# B&R Automation Studio project ABC_Pltzr (part 5)

#### appDraw.typ - Local data types
```iecst
TYPE
	paDrawEnums_typ :
		(
		PADRAW_RECT_MAXIDX := 30
		);
	paCallback_typ : 	STRUCT
		pCallback : REFERENCE TO UDINT;
		callbackValue : UDINT;
		callbackState : UDINT;
		callbackRet : UDINT;
		callbackParams : ARRAY[0..3]OF UDINT;
	END_STRUCT;
	paDrawBoxSize_typ : 	STRUCT
		name : STRING[31];
		length_inch : REAL; (*Width (pixels) of the draw box control*)
		width_inch : REAL; (*Width (pixels) of the draw box control*)
		height_inch : REAL; (*Height (pixels) of the draw box control*)
		length_pixel : UDINT; (*Width (pixels) of the draw box control*)
		width_pixel : UDINT; (*Width (pixels) of the draw box control*)
		height_pixel : UDINT; (*Height (pixels) of the draw box control*)
	END_STRUCT;
	paDrawBoxCtrl_typ : 	STRUCT
		state : UDINT;
		handle : UDINT; (*VISAPI handle returned from VA_Setup()*)
		nameDrawBoxCtrl : STRING[80]; (*DrawBox name for VA_Attach(). It is string with a following format "pageName/LayerName/drawBoxComponentName"*)
		nameVisu : STRING[20]; (*Visualization object name within the project (i.e."Visu", "Panel", "Hmi", etc)*)
		colorIndex : USINT; (*Background color index*)
		width : UDINT; (*Width (pixels) of the draw box control*)
		height : UDINT; (*Height (pixels) of the draw box control*)
	END_STRUCT;
	paDrawTextout_typ : 	STRUCT
		iEnable : USINT; (*Enable text output*)
		iFontIndex : USINT; (*Text font index*)
		iFColorIndex : USINT; (*Text front color index*)
		iBColorIndex : USINT; (*Data line color index*)
		iX : REAL; (*Text x position*)
		iY : REAL; (*Text y poistion*)
		iText : STRING[80]; (*Number of samples in dataset*)
	END_STRUCT;
	paDrawRect_typ : 	STRUCT
		iEnable : USINT; (*Enable text output*)
		iVCHandle : UDINT; (*Text font index*)
		iX : UINT; (*Text x position*)
		iY : UINT; (*Text y poistion*)
		iWidth : UINT; (*Text x position*)
		iHeight : UINT; (*Text y poistion*)
		iFillColorIndex : USINT; (*Text front color index*)
		iBorderColorIndex : USINT; (*Data line color index*)
	END_STRUCT;
	paDrawDataset_typ : 	STRUCT
		iColorIndex : USINT; (*Data line color index*)
		iMinValue : REAL; (*Min value from the data set > will be displayed at 0% on the graph*)
		iMaxValue : REAL; (*Max value from the data set > will be displayed at 100% on the graph*)
		iSizeDataset : UDINT; (*Number of samples in dataset*)
		ipDataset : REFERENCE TO REAL; (*Reference (pointer) to the dataset*)
	END_STRUCT;
	paDrawBoxGrid_typ : 	STRUCT
		ivColorIndex : USINT; (*Grid line color - vertical line*)
		ivLineCount : USINT; (*Number of vertical lines*)
		ivThickRepeat : USINT; (*Place a thicker (i.e. divider) grid line repeat count times - vertical*)
		ihColorIndex : USINT; (*Grid line color - horizontal line*)
		ihLineCount : USINT; (*Number of horizontal lines*)
		ihThickRepeat : USINT; (*Place a thicker (i.e. divider) grid line repeat count times - horizontal*)
	END_STRUCT;
	paDrawXZMotionProfile_typ : 	STRUCT
		ixPhysicalRange : REAL;
		izPhysicalRange : REAL;
		ixPick : REAL;
		izPick : REAL;
		ixDrop : REAL;
		izDrop : REAL;
		iFwdClrIdx : USINT;
		iRevClrIdx : USINT;
		ixCamDataset : paDrawDataset_typ;
		izCamDataset : paDrawDataset_typ;
		idx : UDINT;
		deltaCamMaster : REAL;
		state : UDINT;
	END_STRUCT;
	paDrawBoxDrawing_typ : 	STRUCT
		cb : paCallback_typ;
		ctrl : paDrawBoxCtrl_typ;
		grid : paDrawBoxGrid_typ;
		rect : paDrawRect_typ;
		textout : paDrawTextout_typ;
		data1 : paDrawDataset_typ;
		pRectArray : REFERENCE TO paDrawRect_typ;
		xzProfile : paDrawXZMotionProfile_typ;
	END_STRUCT;
	paCamEditApp_typ : 	STRUCT
		btnPreview : USINT;
		state : UDINT;
		camPointsX : ARRAY[0..3]OF REAL;
		camPointsZ : ARRAY[0..3]OF REAL;
		value : USINT;
	END_STRUCT;
END_TYPE
```

- bgstring.c (reference to Logical/paiComponents/bglib/bgstring.c)

### Program Logical/MachineControl/animation (IEC) - app animation

#### Variables.var
```iecst
VAR
	jj : UDINT := 0;
	ii : UDINT := 0;
END_VAR
```

#### Cyclic.st
```iecst
PROGRAM _CYCLIC
	(* Insert code here *)

	gCtrlAnimation.tmrCase();

	FOR ii :=0 TO 9 BY 1 DO
		IF ii  <  gCtrlAnimation.currentCase THEN
			gCtrlAnimation.visiCase.animationRow[ii] := 0;//visible
		ELSE
			gCtrlAnimation.visiCase.animationRow[ii] := 1;//not visible
		END_IF;

		IF ii  <  gCtrlAnimation.currentRow THEN
			FOR jj := 0 TO 9 BY 1 DO
				IF jj < gConfigApp.options.dryCycleCaseCount THEN
					gCtrlAnimation.visiRow[ii].animationRow[jj] := 0;//visible
				ELSE
					gCtrlAnimation.visiRow[ii].animationRow[jj] := 1;//not visible
				END_IF;
			END_FOR;

		ELSE
			FOR jj := 0 TO 9 BY 1 DO
				gCtrlAnimation.visiRow[ii].animationRow[jj] := 1;//not visible
			END_FOR;
		END_IF;

		IF ii  <  gCtrlAnimation.currentLayer THEN
			FOR jj := 0 TO 9 BY 1 DO
				IF jj < gConfigApp.options.dryCycleRowCount THEN
					gCtrlAnimation.visiLayer[ii].animationRow[jj] := 0;//visible
				ELSE
					gCtrlAnimation.visiLayer[ii].animationRow[jj] := 1;//not visible
				END_IF;
			END_FOR;

		ELSE
			FOR jj := 0 TO 9 BY 1 DO
				gCtrlAnimation.visiLayer[ii].animationRow[jj] := 1;//not visible
			END_FOR;
		END_IF;

	END_FOR;

	IF ((animationState <> 0) AND (NOT gCtrl.main.noFaults)) THEN
		animationState := 50;
	END_IF;

	CASE animationState OF
		0:
			gCtrlAnimation.currentCase := 0;
			gCtrlAnimation.currentRow := 0;
			gCtrlAnimation.currentLayer := 0;
			IF gCtrl.main.modeAuto THEN
				animationState := 10;
				gCtrl.infeedcv.hmiBtnOnOff := 1;
				gCtrl.rowforming.hmiBtnOnOffCV := 1;
			END_IF;
		10:
			gCtrlAnimation.currentCase := gCtrlAnimation.currentCase + 1;
			IF gCtrlAnimation.currentCase >= gConfigApp.options.dryCycleCaseCount THEN
				gCtrl.rowforming.hmiBtnPusherFwd := 1;
				gCtrl.rowforming.hmiBtnPusherRev := 0;
				gCtrl.infeedcv.hmiBtnOnOff := 0;
				gCtrl.rowforming.hmiBtnOnOffCV := 0;
				animationState := 11;
			ELSE
				animationState := 20;
			END_IF;
		11://waiting for row pusher at elev
			IF gCtrl.rowforming.isRowPusherAtElevator THEN
				gCtrlAnimation.currentCase := 0;
				gCtrlAnimation.currentRow := gCtrlAnimation.currentRow + 1;
				gCtrl.rowforming.hmiBtnPusherFwd := 0;
				gCtrl.rowforming.hmiBtnPusherRev := 1;

				IF gCtrlAnimation.currentRow >= gConfigApp.options.dryCycleRowCount THEN
					gCtrl.main.testBit1 := 1;//start elev drycycle
					animationState := 13;
				ELSE
					animationState := 12;
				END_IF;
			END_IF;
		12://waiting for row pusher back home
			IF gCtrl.rowforming.isRowPusherAtHome THEN
				gCtrl.infeedcv.hmiBtnOnOff := 1;
				gCtrl.rowforming.hmiBtnOnOffCV := 1;

				animationState := 20;
			END_IF;
		13:
			IF gCtrl.main.testBit3 THEN//wait for elev dry cycle to complete
				gCtrl.main.testBit3 := 0;
				animationState := 14;
			END_IF;
		14:
			gCtrlAnimation.currentRow := 0;
			gCtrlAnimation.currentLayer := gCtrlAnimation.currentLayer + 1;
			IF gCtrlAnimation.currentLayer >= gConfigApp.options.dryCycleLayerCount THEN
				animationState := 30;
			ELSE
				gCtrl.infeedcv.hmiBtnOnOff := 1;
				gCtrl.rowforming.hmiBtnOnOffCV := 1;

				animationState := 20;
			END_IF;
		20:
			gCtrl.infeedcv.hmiBtnOnOff := 1;
			gCtrl.rowforming.hmiBtnOnOffCV := 1;
			gCtrlAnimation.tmrCase.IN := 0;
			gCtrlAnimation.tmrCase.PT := REAL_TO_UDINT(gConfigApp.options.tmDryCycleCaseTime * 1000);

			IF (gConfigApp.options.dryCycleCaseCount >= 2) AND  (gCtrlAnimation.currentCase = 1) THEN
				gCtrl.caseturner.hmiBtnCaseTurnerUpDown := 1;	//turn on blade1 and case turner
				gCtrl.rowforming.hmiBtnStopBladeUpDown1 := 1;
			ELSE
				gCtrl.caseturner.hmiBtnCaseTurnerUpDown := 0;
				gCtrl.rowforming.hmiBtnStopBladeUpDown1 := 0;
			END_IF;

			animationState := 21;
			IF gCtrl.main.modeManual THEN
				animationState := 50;
			END_IF;

		21:
			gCtrlAnimation.tmrCase.IN := 1;
			IF gCtrlAnimation.tmrCase.Q THEN
				gCtrlAnimation.tmrCase.IN := 0;
				animationState := 10;
			END_IF;

		30:
			//Pallete is Done!
			IF gConfigApp.options.dryCycleLayerDonePause <> 0 THEN
				gPaiHmiRTMenu.iMenuSelectItem[1] := 1;//switch to manual mode
				gCtrlAnimation.tmrCase.IN := 0;
				gCtrlAnimation.tmrCase.PT := T#1s;
				animationState := 31;
			ELSE
				//continue with a new layer
				animationState := 0;//clear all, and start cycle again
			END_IF;
		31:
			gCtrlAnimation.tmrCase.IN := 1;
			IF gCtrlAnimation.tmrCase.Q THEN
				IF gCtrl.main.modeAuto THEN
					animationState := 0;//clear all, and start cycle again
				END_IF;
			END_IF;

		50:
		//wait for resume
			gCtrl.infeedcv.hmiBtnOnOff := 0;
			gCtrl.rowforming.hmiBtnOnOffCV := 0;
			IF gCtrl.main.modeAuto THEN
				gCtrl.infeedcv.hmiBtnOnOff := 1;
				gCtrl.rowforming.hmiBtnOnOffCV := 1;
				animationState := 20;
			END_IF;

	END_CASE;

END_PROGRAM
```

### Program Logical/MachineControl/alarms (IEC) - app alarms

#### Cyclic.ld
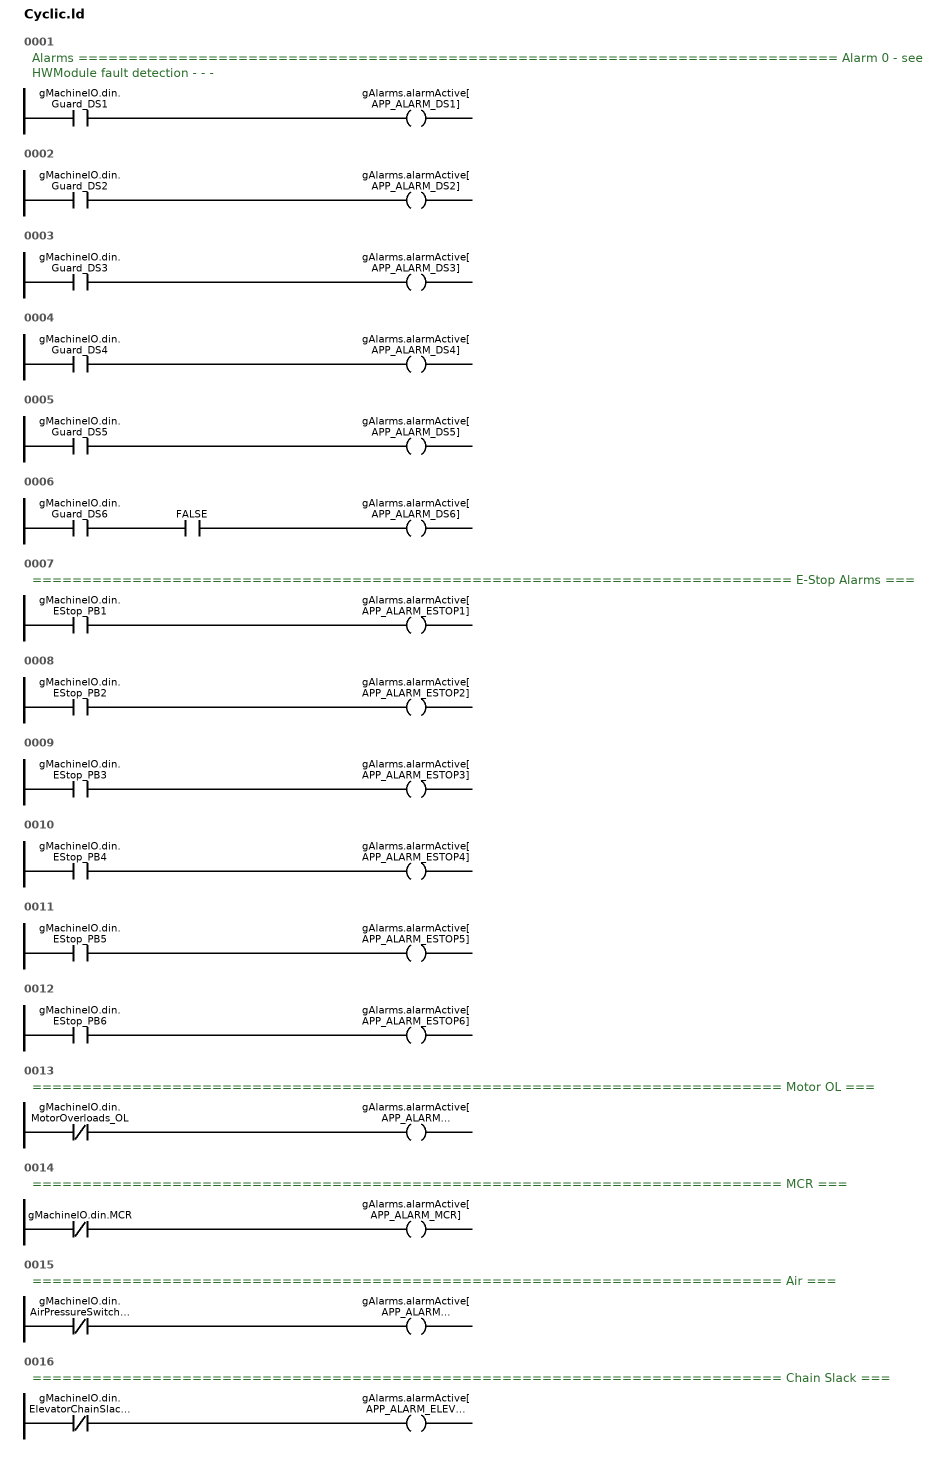
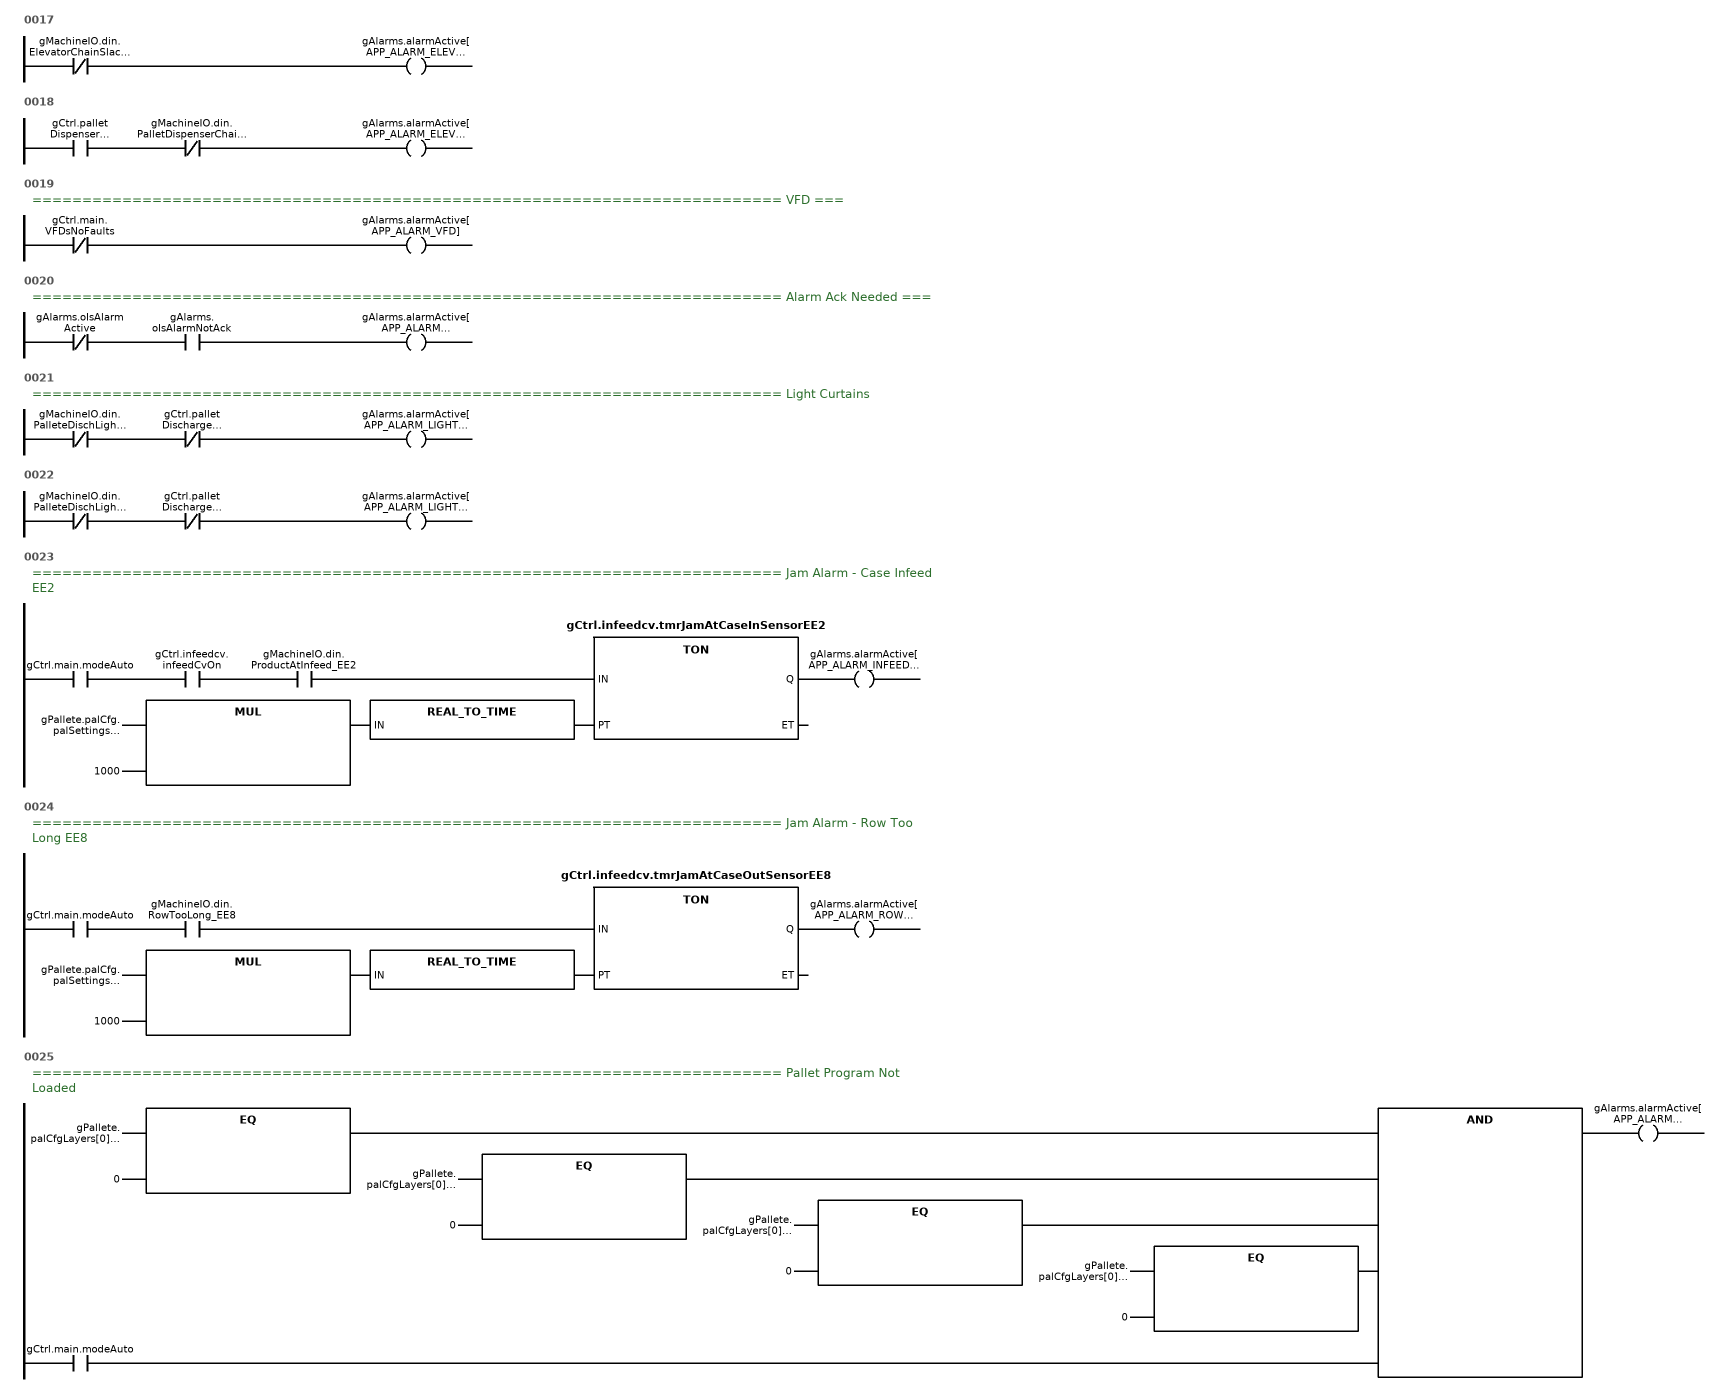
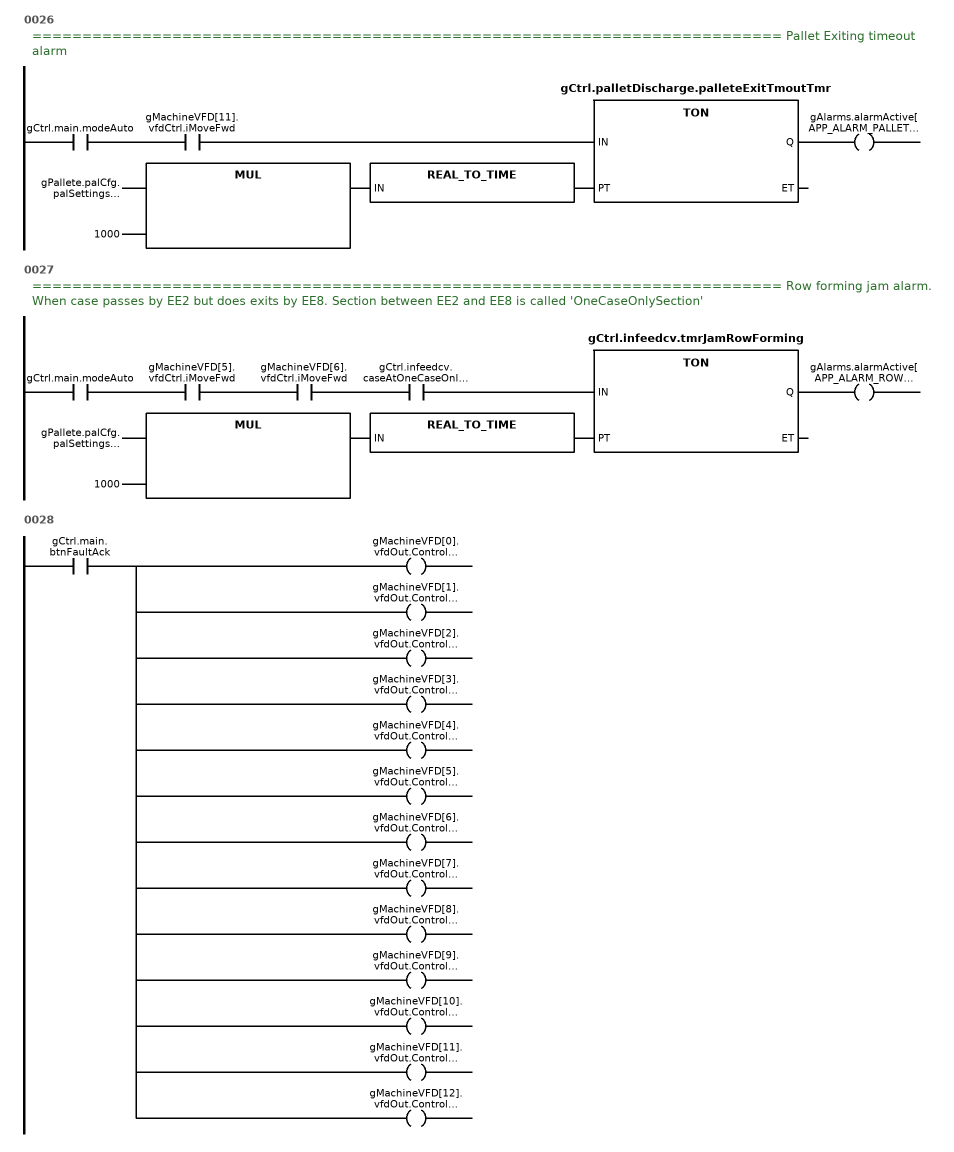
Ladder, written as Structured Text:
```iecst
PROGRAM _CYCLIC
(* Network 1: Alarms ============================================================================ Alarm 0 - see HWModule fault detection - - - *)
gAlarms.alarmActive[APP_ALARM_DS1] := gMachineIO.din.Guard_DS1;

(* Network 2 *)
gAlarms.alarmActive[APP_ALARM_DS2] := gMachineIO.din.Guard_DS2;

(* Network 3 *)
gAlarms.alarmActive[APP_ALARM_DS3] := gMachineIO.din.Guard_DS3;

(* Network 4 *)
gAlarms.alarmActive[APP_ALARM_DS4] := gMachineIO.din.Guard_DS4;

(* Network 5 *)
gAlarms.alarmActive[APP_ALARM_DS5] := gMachineIO.din.Guard_DS5;

(* Network 6 *)
gAlarms.alarmActive[APP_ALARM_DS6] := FALSE;

(* Network 7: ============================================================================ E-Stop Alarms === *)
gAlarms.alarmActive[APP_ALARM_ESTOP1] := gMachineIO.din.EStop_PB1;

(* Network 8 *)
gAlarms.alarmActive[APP_ALARM_ESTOP2] := gMachineIO.din.EStop_PB2;

(* Network 9 *)
gAlarms.alarmActive[APP_ALARM_ESTOP3] := gMachineIO.din.EStop_PB3;

(* Network 10 *)
gAlarms.alarmActive[APP_ALARM_ESTOP4] := gMachineIO.din.EStop_PB4;

(* Network 11 *)
gAlarms.alarmActive[APP_ALARM_ESTOP5] := gMachineIO.din.EStop_PB5;

(* Network 12 *)
gAlarms.alarmActive[APP_ALARM_ESTOP6] := gMachineIO.din.EStop_PB6;

(* Network 13: =========================================================================== Motor OL === *)
gAlarms.alarmActive[APP_ALARM_MOTOROL] := NOT gMachineIO.din.MotorOverloads_OL;

(* Network 14: =========================================================================== MCR === *)
gAlarms.alarmActive[APP_ALARM_MCR] := NOT gMachineIO.din.MCR;

(* Network 15: =========================================================================== Air === *)
gAlarms.alarmActive[APP_ALARM_AIRPRESSURE] := NOT gMachineIO.din.AirPressureSwitch_APS;

(* Network 16: =========================================================================== Chain Slack === *)
gAlarms.alarmActive[APP_ALARM_ELEV_CHAINSLACK_LF] := NOT gMachineIO.din.ElevatorChainSlackLF_LS7;

(* Network 17 *)
gAlarms.alarmActive[APP_ALARM_ELEV_CHAINSLACK_RT] := NOT gMachineIO.din.ElevatorChainSlackRT_LS8;

(* Network 18 *)
gAlarms.alarmActive[APP_ALARM_ELEV_PALLETDISPENS] := gCtrl.palletDispenser.palletDispenserEquipped AND NOT gMachineIO.din.PalletDispenserChainSlack_PR21;

(* Network 19: =========================================================================== VFD === *)
gAlarms.alarmActive[APP_ALARM_VFD] := NOT gCtrl.main.VFDsNoFaults;

(* Network 20: =========================================================================== Alarm Ack Needed === *)
gAlarms.alarmActive[APP_ALARM_ALARMACKNEEDED] := NOT gAlarms.oIsAlarmActive AND gAlarms.oIsAlarmNotAck;

(* Network 21: =========================================================================== Light Curtains *)
gAlarms.alarmActive[APP_ALARM_LIGHT_CURTAIN_OSSD1] := NOT gMachineIO.din.PalleteDischLightCurtain_OSSD1 AND NOT gCtrl.palletDischarge.muteLightCurtainDuringDischarge;

(* Network 22 *)
gAlarms.alarmActive[APP_ALARM_LIGHT_CURTAIN_OSSD2] := NOT gMachineIO.din.PalleteDischLightCurtain_OSSD2 AND NOT gCtrl.palletDischarge.muteLightCurtainDuringDischarge;

(* Network 23: =========================================================================== Jam Alarm - Case Infeed EE2 *)
gCtrl.infeedcv.tmrJamAtCaseInSensorEE2(IN := gCtrl.main.modeAuto AND gCtrl.infeedcv.infeedCvOn AND gMachineIO.din.ProductAtInfeed_EE2, PT := REAL_TO_TIME(gPallete.palCfg.palSettings.timers.JamAlarmTmAtInfeedEE2 * 1000));
gAlarms.alarmActive[APP_ALARM_INFEED_JAM] := gCtrl.infeedcv.tmrJamAtCaseInSensorEE2.Q;

(* Network 24: =========================================================================== Jam Alarm - Row Too Long EE8 *)
gCtrl.infeedcv.tmrJamAtCaseOutSensorEE8(IN := gCtrl.main.modeAuto AND gMachineIO.din.RowTooLong_EE8, PT := REAL_TO_TIME(gPallete.palCfg.palSettings.timers.JamAlarmTmAtRowToLongEE8 * 1000));
gAlarms.alarmActive[APP_ALARM_ROW_TOO_LONG] := gCtrl.infeedcv.tmrJamAtCaseOutSensorEE8.Q;

(* Network 25: =========================================================================== Pallet Program Not Loaded *)
gAlarms.alarmActive[APP_ALARM_INVALID_PROGRAM] := (gPallete.palCfgLayers[0].palCfgRows[0].palCfgCmds[0].cmdCase = 0) AND (gPallete.palCfgLayers[0].palCfgRows[0].palCfgCmds[0].cmdBlade = 0) AND (gPallete.palCfgLayers[0].palCfgRows[0].palCfgCmds[0].cmdFeature = 0) AND (gPallete.palCfgLayers[0].palCfgRows[0].palCfgCmds[0].cmdExtra = 0) AND gCtrl.main.modeAuto;

(* Network 26: =========================================================================== Pallet Exiting timeout alarm *)
gCtrl.palletDischarge.palleteExitTmoutTmr(IN := gCtrl.main.modeAuto AND gMachineVFD[11].vfdCtrl.iMoveFwd, PT := REAL_TO_TIME(gPallete.palCfg.palSettings.timers.palletExitAlarmTm * 1000));
gAlarms.alarmActive[APP_ALARM_PALLET_EXIT_TIMEOUT] := gCtrl.palletDischarge.palleteExitTmoutTmr.Q;

(* Network 27: =========================================================================== Row forming jam alarm. When case passes by EE2 but does exits by EE8. Section between EE2 and EE8 is called 'OneCaseOnlySection' *)
gCtrl.infeedcv.tmrJamRowForming(IN := gCtrl.main.modeAuto AND gMachineVFD[5].vfdCtrl.iMoveFwd AND gMachineVFD[6].vfdCtrl.iMoveFwd AND gCtrl.infeedcv.caseAtOneCaseOnlySection, PT := REAL_TO_TIME(gPallete.palCfg.palSettings.timers.JamAlarmTmRowForming * 1000));
gAlarms.alarmActive[APP_ALARM_ROW_FORMING_JAM] := gCtrl.infeedcv.tmrJamRowForming.Q;

(* Network 28 *)
gMachineVFD[0].vfdOut.Control.FaultReset := gCtrl.main.btnFaultAck;
gMachineVFD[1].vfdOut.Control.FaultReset := gCtrl.main.btnFaultAck;
gMachineVFD[2].vfdOut.Control.FaultReset := gCtrl.main.btnFaultAck;
gMachineVFD[3].vfdOut.Control.FaultReset := gCtrl.main.btnFaultAck;
gMachineVFD[4].vfdOut.Control.FaultReset := gCtrl.main.btnFaultAck;
gMachineVFD[5].vfdOut.Control.FaultReset := gCtrl.main.btnFaultAck;
gMachineVFD[6].vfdOut.Control.FaultReset := gCtrl.main.btnFaultAck;
gMachineVFD[7].vfdOut.Control.FaultReset := gCtrl.main.btnFaultAck;
gMachineVFD[8].vfdOut.Control.FaultReset := gCtrl.main.btnFaultAck;
gMachineVFD[9].vfdOut.Control.FaultReset := gCtrl.main.btnFaultAck;
gMachineVFD[10].vfdOut.Control.FaultReset := gCtrl.main.btnFaultAck;
gMachineVFD[11].vfdOut.Control.FaultReset := gCtrl.main.btnFaultAck;
gMachineVFD[12].vfdOut.Control.FaultReset := gCtrl.main.btnFaultAck;
END_PROGRAM
```

### Program Logical/MachineControl/messages (IEC) - app HMI messages

#### Cyclic.ld
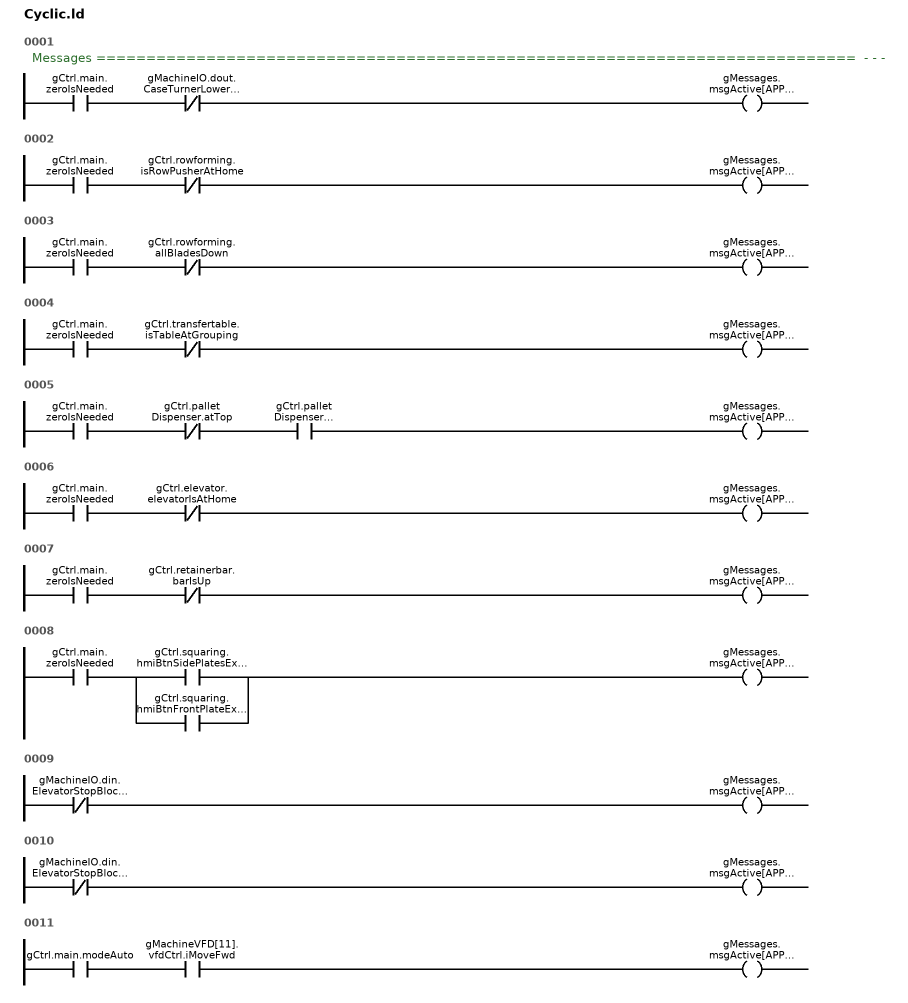
Ladder, written as Structured Text:
```iecst
PROGRAM _CYCLIC
(* Network 1: Messages ============================================================================  - - - *)
gMessages.msgActive[APP_MSG_ZERO_CASETURNER] := gCtrl.main.zeroIsNeeded AND NOT gMachineIO.dout.CaseTurnerLower_SOL2B;

(* Network 2 *)
gMessages.msgActive[APP_MSG_ZERO_ROWPUSHER] := gCtrl.main.zeroIsNeeded AND NOT gCtrl.rowforming.isRowPusherAtHome;

(* Network 3 *)
gMessages.msgActive[APP_MSG_ZERO_BLADESTOP] := gCtrl.main.zeroIsNeeded AND NOT gCtrl.rowforming.allBladesDown;

(* Network 4 *)
gMessages.msgActive[APP_MSG_ZERO_TABLE] := gCtrl.main.zeroIsNeeded AND NOT gCtrl.transfertable.isTableAtGrouping;

(* Network 5 *)
gMessages.msgActive[APP_MSG_ZERO_PALLETELIFT] := gCtrl.main.zeroIsNeeded AND NOT gCtrl.palletDispenser.atTop AND gCtrl.palletDispenser.palletDispenserEquipped;

(* Network 6 *)
gMessages.msgActive[APP_MSG_ZERO_ELEVATOR] := gCtrl.main.zeroIsNeeded AND NOT gCtrl.elevator.elevatorIsAtHome;

(* Network 7 *)
gMessages.msgActive[APP_MSG_ZERO_RETAINERBAR] := gCtrl.main.zeroIsNeeded AND NOT gCtrl.retainerbar.barIsUp;

(* Network 8 *)
gMessages.msgActive[APP_MSG_ZERO_SQUARING] := gCtrl.main.zeroIsNeeded AND (gCtrl.squaring.hmiBtnSidePlatesExtRet OR gCtrl.squaring.hmiBtnFrontPlateExtRet);

(* Network 9 *)
gMessages.msgActive[APP_MSG_STOP_BLOCK_LF] := NOT gMachineIO.din.ElevatorStopBlockLF_PR33;

(* Network 10 *)
gMessages.msgActive[APP_MSG_STOP_BLOCK_RT] := NOT gMachineIO.din.ElevatorStopBlockRT_PR34;

(* Network 11 *)
gMessages.msgActive[APP_MSG_PALLETE_EXITING] := gCtrl.main.modeAuto AND gMachineVFD[11].vfdCtrl.iMoveFwd;
END_PROGRAM
```

### Program Logical/MachineControl/safety (IEC) - app Machine Safety

#### Cyclic.ld
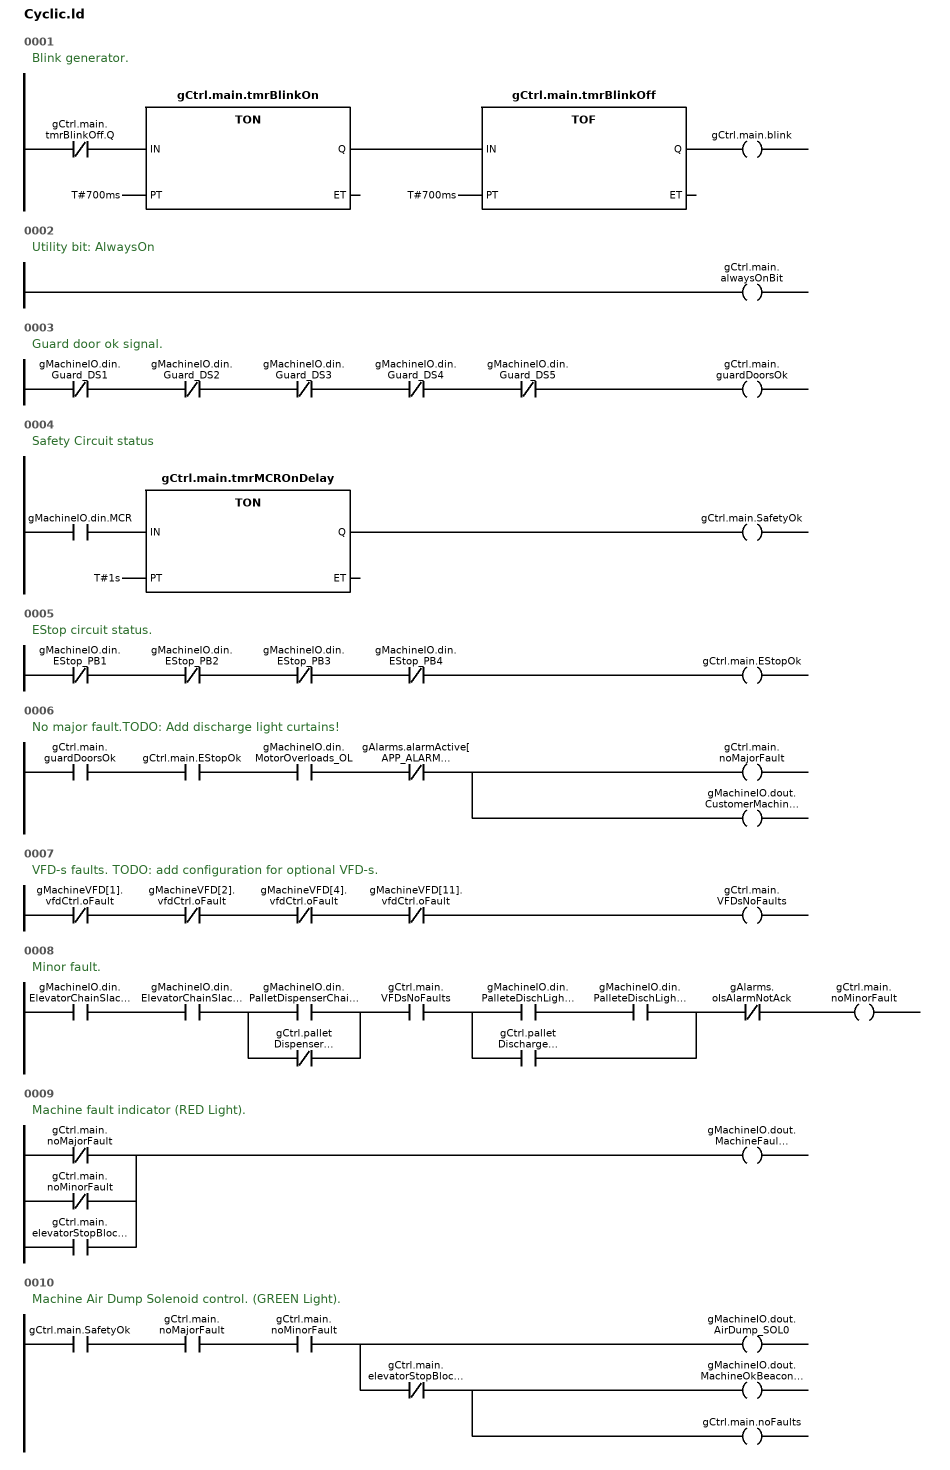
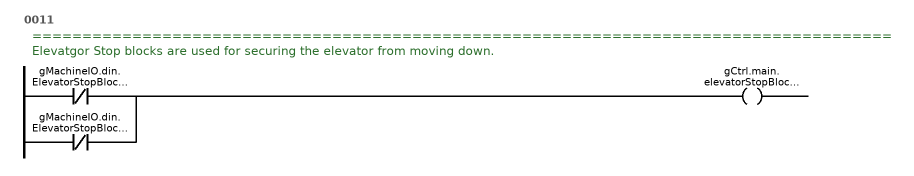
Ladder, written as Structured Text:
```iecst
PROGRAM _CYCLIC
VAR
    _p1 : BOOL;
    _p2 : BOOL;
    _p3 : BOOL;
    _p4 : BOOL;
END_VAR
(* Network 1: Blink generator. *)
gCtrl.main.tmrBlinkOn(IN := NOT gCtrl.main.tmrBlinkOff.Q, PT := T#700ms);
gCtrl.main.tmrBlinkOff(IN := gCtrl.main.tmrBlinkOn.Q, PT := T#700ms);
gCtrl.main.blink := gCtrl.main.tmrBlinkOff.Q;

(* Network 2: Utility bit: AlwaysOn *)
gCtrl.main.alwaysOnBit := TRUE;

(* Network 3: Guard door ok signal. *)
gCtrl.main.guardDoorsOk := NOT gMachineIO.din.Guard_DS1 AND NOT gMachineIO.din.Guard_DS2 AND NOT gMachineIO.din.Guard_DS3 AND NOT gMachineIO.din.Guard_DS4 AND NOT gMachineIO.din.Guard_DS5;

(* Network 4: Safety Circuit status *)
gCtrl.main.tmrMCROnDelay(IN := gMachineIO.din.MCR, PT := T#1s);
gCtrl.main.SafetyOk := gCtrl.main.tmrMCROnDelay.Q;

(* Network 5: EStop circuit status. *)
gCtrl.main.EStopOk := NOT gMachineIO.din.EStop_PB1 AND NOT gMachineIO.din.EStop_PB2 AND NOT gMachineIO.din.EStop_PB3 AND NOT gMachineIO.din.EStop_PB4;

(* Network 6: No major fault.TODO: Add discharge light curtains! *)
_p1 := gCtrl.main.guardDoorsOk AND gCtrl.main.EStopOk AND gMachineIO.din.MotorOverloads_OL AND NOT gAlarms.alarmActive[APP_ALARM_HWMODULE];
gCtrl.main.noMajorFault := _p1;
gMachineIO.dout.CustomerMachineRunning_CR5 := _p1;

(* Network 7: VFD-s faults. TODO: add configuration for optional VFD-s. *)
gCtrl.main.VFDsNoFaults := NOT gMachineVFD[1].vfdCtrl.oFault AND NOT gMachineVFD[2].vfdCtrl.oFault AND NOT gMachineVFD[4].vfdCtrl.oFault AND NOT gMachineVFD[11].vfdCtrl.oFault;

(* Network 8: Minor fault. *)
_p2 := gMachineIO.din.ElevatorChainSlackLF_LS7 AND gMachineIO.din.ElevatorChainSlackRT_LS8;
_p3 := _p2 AND (gMachineIO.din.PalletDispenserChainSlack_PR21 OR NOT gCtrl.palletDispenser.palletDispenserEquipped) AND gCtrl.main.VFDsNoFaults;
gCtrl.main.noMinorFault := _p3 AND ((gMachineIO.din.PalleteDischLightCurtain_OSSD1 AND gMachineIO.din.PalleteDischLightCurtain_OSSD2) OR gCtrl.palletDischarge.muteLightCurtainDuringDischarge) AND NOT gAlarms.oIsAlarmNotAck;

(* Network 9: Machine fault indicator (RED Light). *)
gMachineIO.dout.MachineFaultBeacon_LT1 := NOT gCtrl.main.noMajorFault OR NOT gCtrl.main.noMinorFault OR gCtrl.main.elevatorStopBlockActive;

(* Network 10: Machine Air Dump Solenoid control. (GREEN Light). *)
_p4 := gCtrl.main.SafetyOk AND gCtrl.main.noMajorFault AND gCtrl.main.noMinorFault;
gMachineIO.dout.AirDump_SOL0 := _p4;
gMachineIO.dout.MachineOkBeacon_LT2 := _p4 AND NOT gCtrl.main.elevatorStopBlockActive;
gCtrl.main.noFaults := _p4 AND NOT gCtrl.main.elevatorStopBlockActive;

(* Network 11: ====================================================================================== Elevatgor Stop blocks are used for securing the elevator from moving down. *)
gCtrl.main.elevatorStopBlockActive := NOT gMachineIO.din.ElevatorStopBlockLF_PR33 OR NOT gMachineIO.din.ElevatorStopBlockRT_PR34;
END_PROGRAM
```

### Program Logical/MachineControl/machzero (IEC) - app Machine Zeroing

#### Cyclic.ld
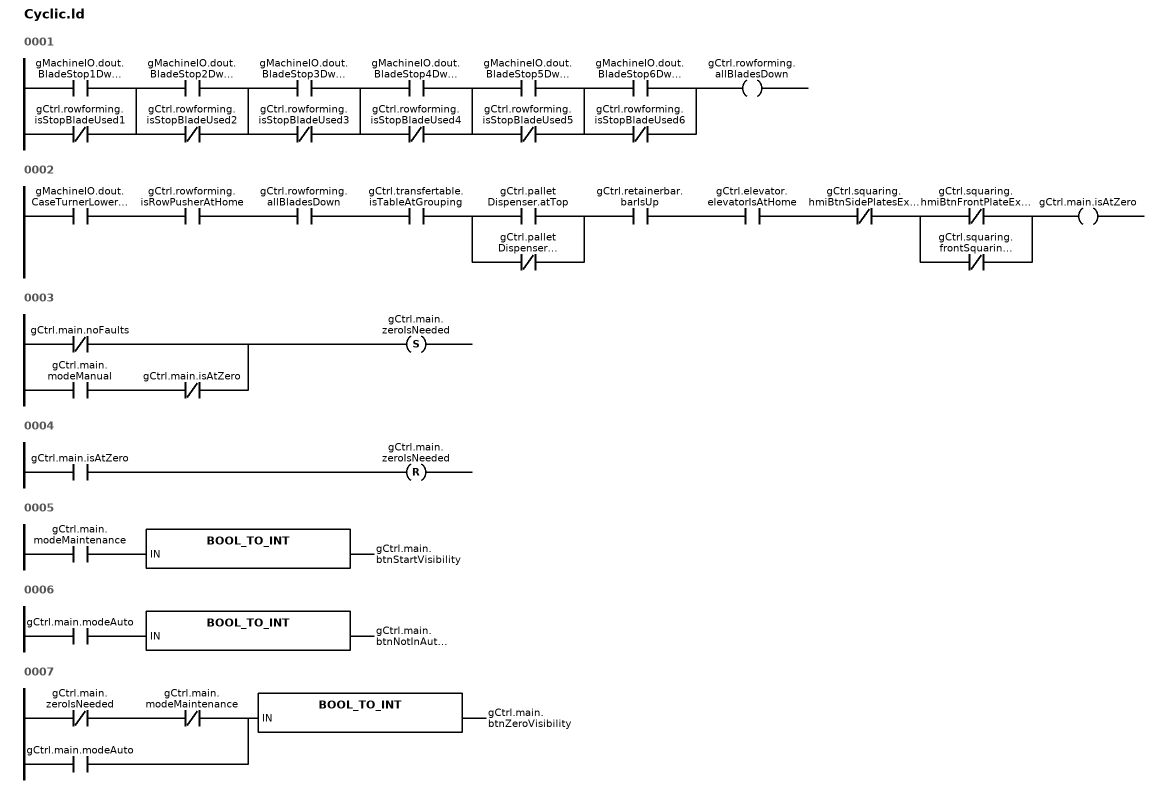
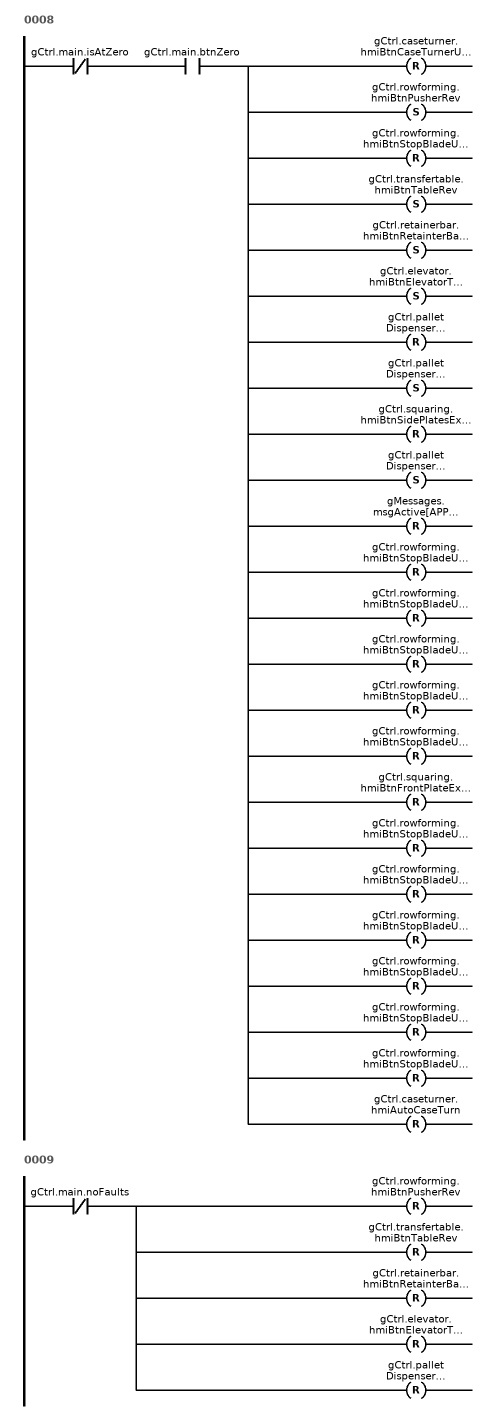
Ladder, written as Structured Text:
```iecst
PROGRAM _CYCLIC
VAR
    _p1 : BOOL;
    _p2 : BOOL;
    _p3 : BOOL;
    _p4 : BOOL;
    _p5 : BOOL;
    _p6 : BOOL;
    _p7 : BOOL;
    _p8 : BOOL;
    _p9 : BOOL;
    _p10 : BOOL;
    _p11 : BOOL;
    _p12 : BOOL;
END_VAR
(* Network 1 *)
_p1 := (gMachineIO.dout.BladeStop1Dw_SOL3B OR NOT gCtrl.rowforming.isStopBladeUsed1) AND gMachineIO.dout.BladeStop2Dw_SOL4B;
_p2 := (gMachineIO.dout.BladeStop1Dw_SOL3B OR NOT gCtrl.rowforming.isStopBladeUsed1) AND NOT gCtrl.rowforming.isStopBladeUsed2;
_p3 := (_p1 OR _p2) AND gMachineIO.dout.BladeStop3Dw_SOL5B;
_p4 := (_p1 OR _p2) AND NOT gCtrl.rowforming.isStopBladeUsed3;
_p5 := (_p3 OR _p4) AND gMachineIO.dout.BladeStop4Dw_SOL6B;
_p6 := (_p3 OR _p4) AND NOT gCtrl.rowforming.isStopBladeUsed4;
_p7 := (_p5 OR _p6) AND gMachineIO.dout.BladeStop5Dw_SOL13B;
_p8 := (_p5 OR _p6) AND NOT gCtrl.rowforming.isStopBladeUsed5;
gCtrl.rowforming.allBladesDown := (_p7 OR _p8) AND (gMachineIO.dout.BladeStop6Dw_SOL14B OR NOT gCtrl.rowforming.isStopBladeUsed6);

(* Network 2 *)
_p9 := gMachineIO.dout.CaseTurnerLower_SOL2B AND gCtrl.rowforming.isRowPusherAtHome AND gCtrl.rowforming.allBladesDown AND gCtrl.transfertable.isTableAtGrouping;
_p10 := _p9 AND (gCtrl.palletDispenser.atTop OR NOT gCtrl.palletDispenser.palletDispenserEquipped) AND gCtrl.retainerbar.barIsUp AND gCtrl.elevator.elevatorIsAtHome AND NOT gCtrl.squaring.hmiBtnSidePlatesExtRet;
gCtrl.main.isAtZero := _p10 AND (NOT gCtrl.squaring.hmiBtnFrontPlateExtRet OR NOT gCtrl.squaring.frontSquaringEquipped);

(* Network 3 *)
IF NOT gCtrl.main.noFaults OR (gCtrl.main.modeManual AND NOT gCtrl.main.isAtZero) THEN
    gCtrl.main.zeroIsNeeded := TRUE;
END_IF;

(* Network 4 *)
IF gCtrl.main.isAtZero THEN gCtrl.main.zeroIsNeeded := FALSE; END_IF;

(* Network 5 *)
gCtrl.main.btnStartVisibility := BOOL_TO_INT(gCtrl.main.modeMaintenance);

(* Network 6 *)
gCtrl.main.btnNotInAutoModeVisibility := BOOL_TO_INT(gCtrl.main.modeAuto);

(* Network 7 *)
gCtrl.main.btnZeroVisibility := BOOL_TO_INT((NOT gCtrl.main.zeroIsNeeded AND NOT gCtrl.main.modeMaintenance) OR gCtrl.main.modeAuto);

(* Network 8 *)
_p11 := NOT gCtrl.main.isAtZero AND gCtrl.main.btnZero;
IF NOT gCtrl.main.isAtZero AND gCtrl.main.btnZero THEN
    gCtrl.caseturner.hmiBtnCaseTurnerUpDown := FALSE;
END_IF;
IF _p11 THEN
    gCtrl.rowforming.hmiBtnPusherRev := TRUE;
    gCtrl.rowforming.hmiBtnStopBladeUpDown1 := FALSE;
    gCtrl.transfertable.hmiBtnTableRev := TRUE;
    gCtrl.retainerbar.hmiBtnRetainterBarRev := TRUE;
    gCtrl.elevator.hmiBtnElevatorToGrouping := TRUE;
    gCtrl.palletDispenser.hmiBtnPalletClawsOpenClose := FALSE;
    gCtrl.palletDispenser.hmiBtnClawsLiftToTop := TRUE;
    gCtrl.squaring.hmiBtnSidePlatesExtRet := FALSE;
    gCtrl.palletDispenser.hmiBtnPalletClawsOpenClose := TRUE;
    gMessages.msgActive[APP_MSG_PALLETE_COMPLETE] := FALSE;
    gCtrl.rowforming.hmiBtnStopBladeUpDown2 := FALSE;
    gCtrl.rowforming.hmiBtnStopBladeUpDown3 := FALSE;
    gCtrl.rowforming.hmiBtnStopBladeUpDown4 := FALSE;
    gCtrl.rowforming.hmiBtnStopBladeUpDown5 := FALSE;
    gCtrl.rowforming.hmiBtnStopBladeUpDown6 := FALSE;
    gCtrl.squaring.hmiBtnFrontPlateExtRet := FALSE;
    gCtrl.rowforming.hmiBtnStopBladeUpDownQuick1 := FALSE;
    gCtrl.rowforming.hmiBtnStopBladeUpDownQuick2 := FALSE;
    gCtrl.rowforming.hmiBtnStopBladeUpDownQuick3 := FALSE;
    gCtrl.rowforming.hmiBtnStopBladeUpDownQuick4 := FALSE;
    gCtrl.rowforming.hmiBtnStopBladeUpDownQuick5 := FALSE;
    gCtrl.rowforming.hmiBtnStopBladeUpDownQuick6 := FALSE;
    gCtrl.caseturner.hmiAutoCaseTurn := FALSE;
END_IF;

(* Network 9 *)
_p12 := NOT gCtrl.main.noFaults;
IF NOT gCtrl.main.noFaults THEN gCtrl.rowforming.hmiBtnPusherRev := FALSE; END_IF;
IF _p12 THEN
    gCtrl.transfertable.hmiBtnTableRev := FALSE;
    gCtrl.retainerbar.hmiBtnRetainterBarRev := FALSE;
    gCtrl.elevator.hmiBtnElevatorToGrouping := FALSE;
    gCtrl.palletDispenser.hmiBtnClawsLiftToTop := FALSE;
END_IF;
END_PROGRAM
```

- Program Logical/MachineControl/infcvidle (IEC) - app infeed CV idle logic (no source held here)

### Program Logical/MachineControl/rowforming (IEC) - app row forming

#### Cyclic.ld - Cyclic code
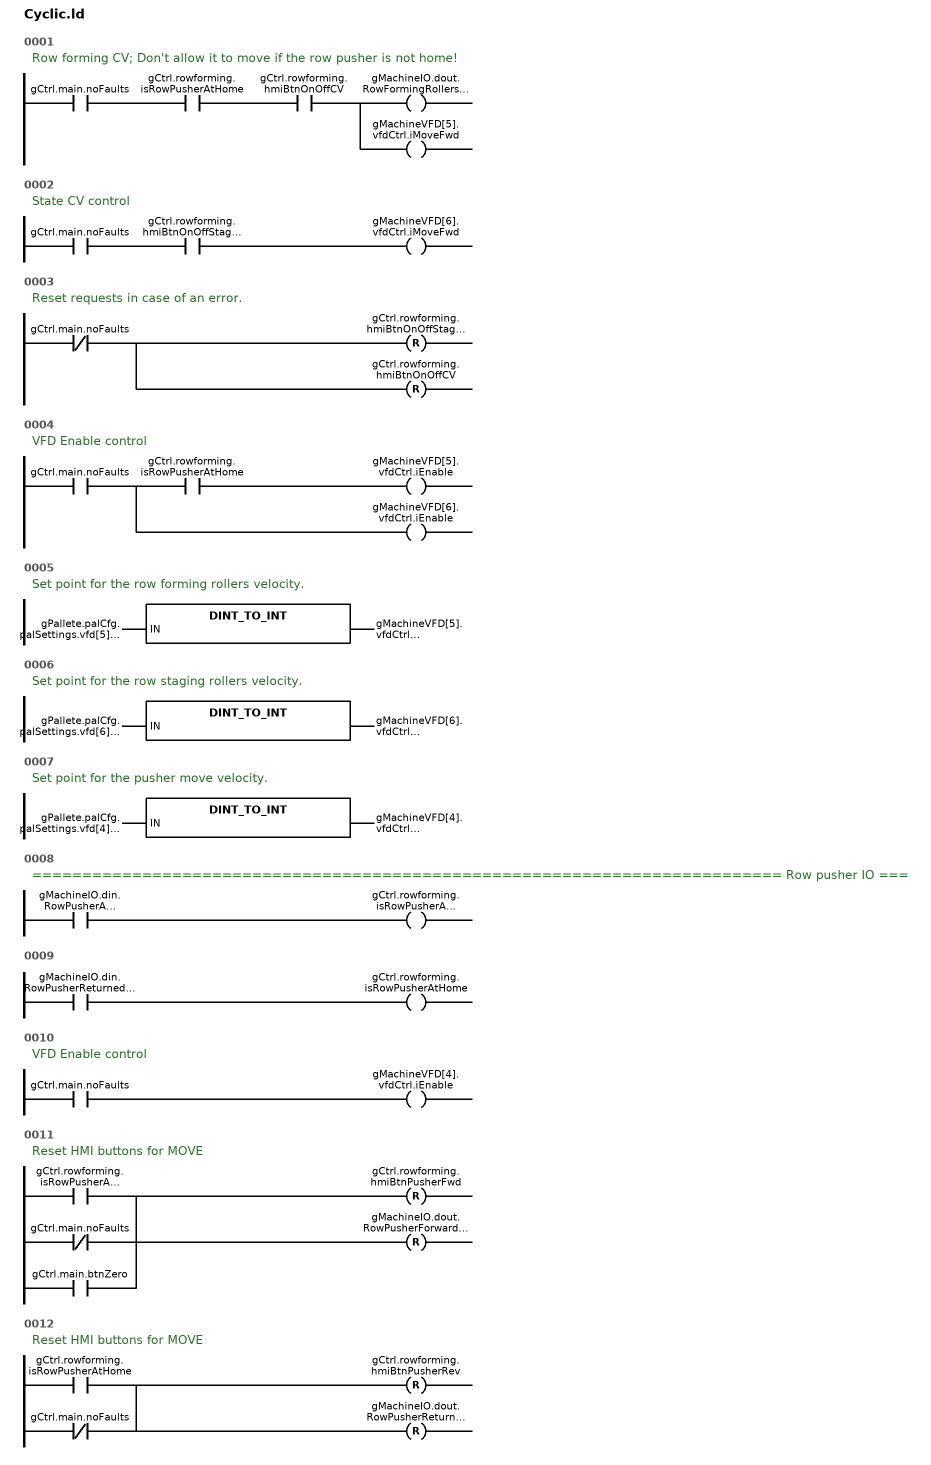
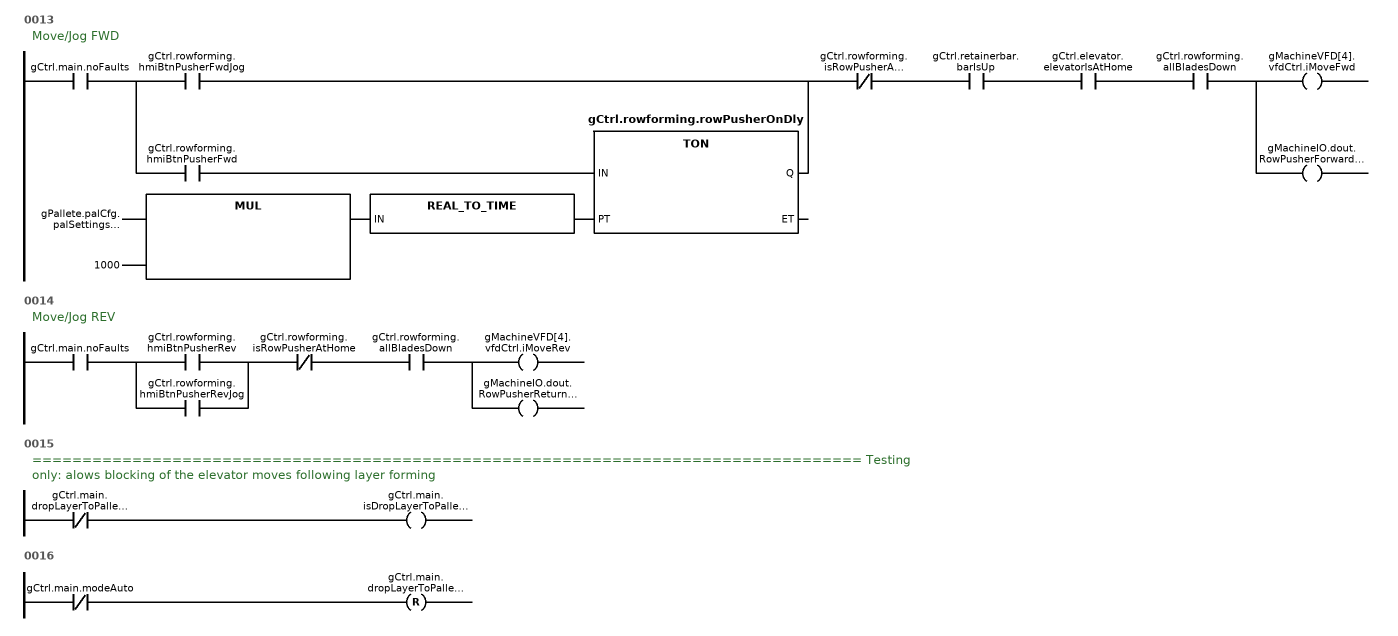
Ladder, written as Structured Text:
```iecst
PROGRAM _CYCLIC
VAR
    _p1 : BOOL;
    _p2 : BOOL;
    _p3 : BOOL;
    _p4 : BOOL;
    _p5 : BOOL;
    _p6 : BOOL;
    _p7 : BOOL;
    _p8 : BOOL;
    _p9 : BOOL;
END_VAR
(* Network 1: Row forming CV; Don't allow it to move if the row pusher is not home! *)
_p1 := gCtrl.main.noFaults AND gCtrl.rowforming.isRowPusherAtHome AND gCtrl.rowforming.hmiBtnOnOffCV;
gMachineIO.dout.RowFormingRollers_M5 := _p1;
gMachineVFD[5].vfdCtrl.iMoveFwd := _p1;

(* Network 2: State CV control *)
gMachineVFD[6].vfdCtrl.iMoveFwd := gCtrl.main.noFaults AND gCtrl.rowforming.hmiBtnOnOffStageCV;

(* Network 3: Reset requests in case of an error. *)
_p2 := NOT gCtrl.main.noFaults;
IF NOT gCtrl.main.noFaults THEN gCtrl.rowforming.hmiBtnOnOffStageCV := FALSE; END_IF;
IF _p2 THEN gCtrl.rowforming.hmiBtnOnOffCV := FALSE; END_IF;

(* Network 4: VFD Enable control *)
gMachineVFD[5].vfdCtrl.iEnable := gCtrl.main.noFaults AND gCtrl.rowforming.isRowPusherAtHome;
gMachineVFD[6].vfdCtrl.iEnable := gCtrl.main.noFaults;

(* Network 5: Set point for the row forming rollers velocity. *)
gMachineVFD[5].vfdCtrl.iVelocitySetPoint := DINT_TO_INT(gPallete.palCfg.palSettings.vfd[5].velocity_rpm);

(* Network 6: Set point for the row staging rollers velocity. *)
gMachineVFD[6].vfdCtrl.iVelocitySetPoint := DINT_TO_INT(gPallete.palCfg.palSettings.vfd[6].velocity_rpm);

(* Network 7: Set point for the pusher move velocity. *)
gMachineVFD[4].vfdCtrl.iVelocitySetPoint := DINT_TO_INT(gPallete.palCfg.palSettings.vfd[4].velocity_rpm);

(* Network 8: =========================================================================== Row pusher IO === *)
gCtrl.rowforming.isRowPusherAtElevator := gMachineIO.din.RowPusherAtElevator_PR13;

(* Network 9 *)
gCtrl.rowforming.isRowPusherAtHome := gMachineIO.din.RowPusherReturned_PR11;

(* Network 10: VFD Enable control *)
gMachineVFD[4].vfdCtrl.iEnable := gCtrl.main.noFaults;

(* Network 11: Reset HMI buttons for MOVE *)
_p3 := gCtrl.rowforming.isRowPusherAtElevator;
_p4 := NOT gCtrl.main.noFaults;
_p5 := gCtrl.main.btnZero;
IF gCtrl.rowforming.isRowPusherAtElevator OR NOT gCtrl.main.noFaults OR gCtrl.main.btnZero THEN
    gCtrl.rowforming.hmiBtnPusherFwd := FALSE;
END_IF;
IF _p3 OR _p4 OR _p5 THEN gMachineIO.dout.RowPusherForward_M4F := FALSE; END_IF;

(* Network 12: Reset HMI buttons for MOVE *)
_p6 := gCtrl.rowforming.isRowPusherAtHome;
_p7 := NOT gCtrl.main.noFaults;
IF gCtrl.rowforming.isRowPusherAtHome OR NOT gCtrl.main.noFaults THEN
    gCtrl.rowforming.hmiBtnPusherRev := FALSE;
END_IF;
IF _p6 OR _p7 THEN gMachineIO.dout.RowPusherReturn_M4R := FALSE; END_IF;

(* Network 13: Move/Jog FWD *)
_p8 := ((gCtrl.main.noFaults AND gCtrl.rowforming.hmiBtnPusherFwdJog) OR gCtrl.rowforming.rowPusherOnDly.Q) AND NOT gCtrl.rowforming.isRowPusherAtElevator AND gCtrl.retainerbar.barIsUp AND gCtrl.elevator.elevatorIsAtHome AND gCtrl.rowforming.allBladesDown;
gMachineVFD[4].vfdCtrl.iMoveFwd := _p8;
gCtrl.rowforming.rowPusherOnDly(IN := gCtrl.main.noFaults AND gCtrl.rowforming.hmiBtnPusherFwd, PT := REAL_TO_TIME(gPallete.palCfg.palSettings.timers.dlyRowDoneToRowPush * 1000));
gMachineIO.dout.RowPusherForward_M4F := _p8;

(* Network 14: Move/Jog REV *)
_p9 := gCtrl.main.noFaults AND (gCtrl.rowforming.hmiBtnPusherRev OR gCtrl.rowforming.hmiBtnPusherRevJog) AND NOT gCtrl.rowforming.isRowPusherAtHome AND gCtrl.rowforming.allBladesDown;
gMachineVFD[4].vfdCtrl.iMoveRev := _p9;
gMachineIO.dout.RowPusherReturn_M4R := _p9;

(* Network 15: =================================================================================== Testing only: alows blocking of the elevator moves following layer forming *)
gCtrl.main.isDropLayerToPalletAllowed := NOT gCtrl.main.dropLayerToPalletBlock;

(* Network 16 *)
IF NOT gCtrl.main.modeAuto THEN gCtrl.main.dropLayerToPalletBlock := FALSE; END_IF;
END_PROGRAM
```

### Program Logical/MachineControl/transtable (IEC) - app transfer table

#### Cyclic.ld
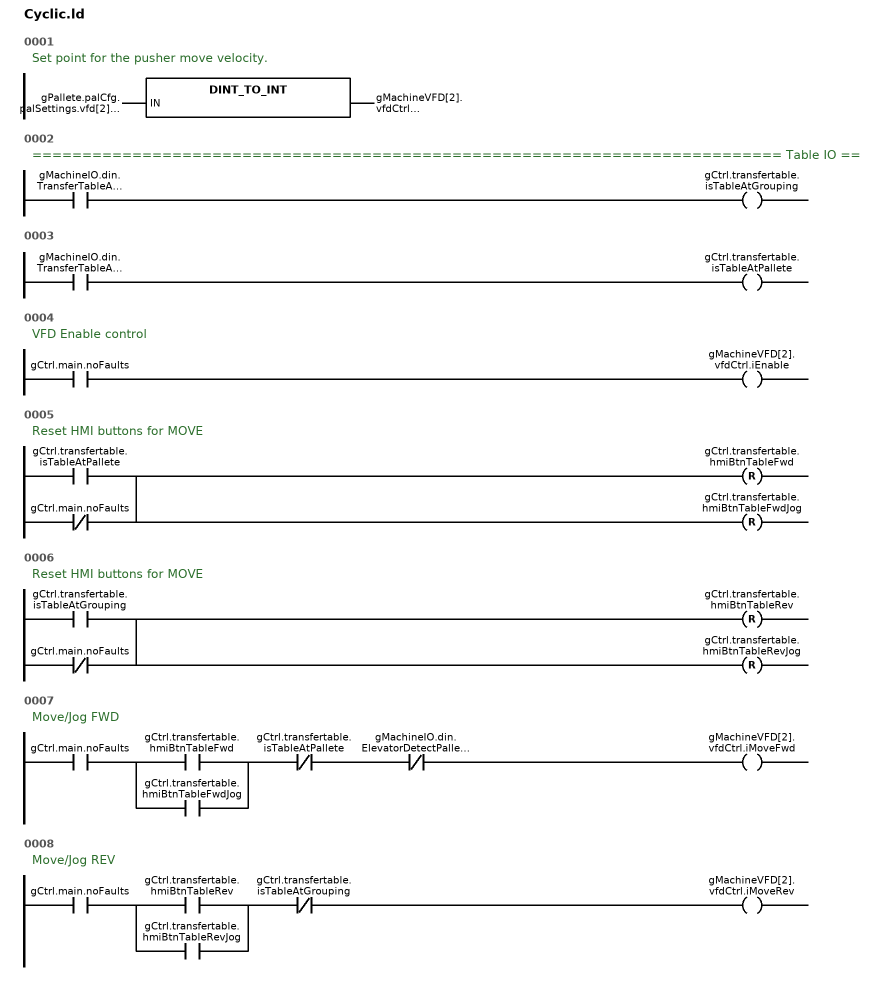
Ladder, written as Structured Text:
```iecst
PROGRAM _CYCLIC
VAR
    _p1 : BOOL;
    _p2 : BOOL;
    _p3 : BOOL;
    _p4 : BOOL;
END_VAR
(* Network 1: Set point for the pusher move velocity. *)
gMachineVFD[2].vfdCtrl.iVelocitySetPoint := DINT_TO_INT(gPallete.palCfg.palSettings.vfd[2].velocity_rpm);

(* Network 2: =========================================================================== Table IO == *)
gCtrl.transfertable.isTableAtGrouping := gMachineIO.din.TransferTableAtGrouping_PR6;

(* Network 3 *)
gCtrl.transfertable.isTableAtPallete := gMachineIO.din.TransferTableAtPallete_PR5;

(* Network 4: VFD Enable control *)
gMachineVFD[2].vfdCtrl.iEnable := gCtrl.main.noFaults;

(* Network 5: Reset HMI buttons for MOVE *)
_p1 := gCtrl.transfertable.isTableAtPallete;
_p2 := NOT gCtrl.main.noFaults;
IF gCtrl.transfertable.isTableAtPallete OR NOT gCtrl.main.noFaults THEN
    gCtrl.transfertable.hmiBtnTableFwd := FALSE;
END_IF;
IF _p1 OR _p2 THEN gCtrl.transfertable.hmiBtnTableFwdJog := FALSE; END_IF;

(* Network 6: Reset HMI buttons for MOVE *)
_p3 := gCtrl.transfertable.isTableAtGrouping;
_p4 := NOT gCtrl.main.noFaults;
IF gCtrl.transfertable.isTableAtGrouping OR NOT gCtrl.main.noFaults THEN
    gCtrl.transfertable.hmiBtnTableRev := FALSE;
END_IF;
IF _p3 OR _p4 THEN gCtrl.transfertable.hmiBtnTableRevJog := FALSE; END_IF;

(* Network 7: Move/Jog FWD *)
gMachineVFD[2].vfdCtrl.iMoveFwd := gCtrl.main.noFaults AND (gCtrl.transfertable.hmiBtnTableFwd OR gCtrl.transfertable.hmiBtnTableFwdJog) AND NOT gCtrl.transfertable.isTableAtPallete AND NOT gMachineIO.din.ElevatorDetectPalletLayerLF_EE1;

(* Network 8: Move/Jog REV *)
gMachineVFD[2].vfdCtrl.iMoveRev := gCtrl.main.noFaults AND (gCtrl.transfertable.hmiBtnTableRev OR gCtrl.transfertable.hmiBtnTableRevJog) AND NOT gCtrl.transfertable.isTableAtGrouping;
END_PROGRAM
```

### Program Logical/MachineControl/palletinfcv (IEC) - app pallet infeed conveyer

#### Cyclic.ld
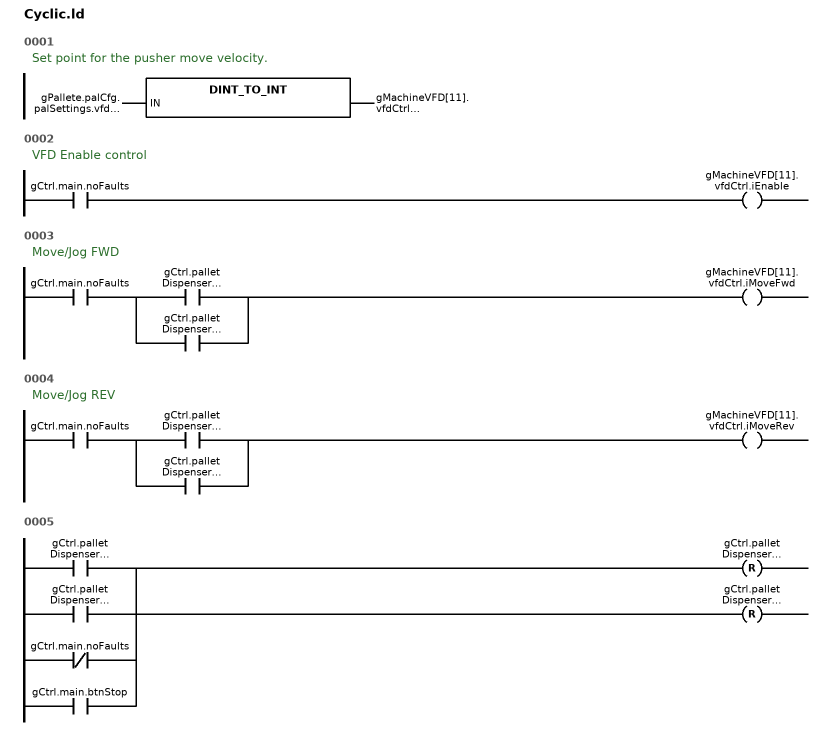
Ladder, written as Structured Text:
```iecst
PROGRAM _CYCLIC
VAR
    _p1 : BOOL;
    _p2 : BOOL;
    _p3 : BOOL;
    _p4 : BOOL;
END_VAR
(* Network 1: Set point for the pusher move velocity. *)
gMachineVFD[11].vfdCtrl.iVelocitySetPoint := DINT_TO_INT(gPallete.palCfg.palSettings.vfd[11].velocity_rpm);

(* Network 2: VFD Enable control *)
gMachineVFD[11].vfdCtrl.iEnable := gCtrl.main.noFaults;

(* Network 3: Move/Jog FWD *)
gMachineVFD[11].vfdCtrl.iMoveFwd := gCtrl.main.noFaults AND (gCtrl.palletDispenser.hmiBtnPalletInCVFwd OR gCtrl.palletDispenser.hmiBtnPalletInCVFwdJog);

(* Network 4: Move/Jog REV *)
gMachineVFD[11].vfdCtrl.iMoveRev := gCtrl.main.noFaults AND (gCtrl.palletDispenser.hmiBtnPalletInCVRev OR gCtrl.palletDispenser.hmiBtnPalletInCVRevJog);

(* Network 5 *)
_p1 := gCtrl.palletDispenser.hmiBtnPalletInCVRevJog;
_p2 := gCtrl.palletDispenser.hmiBtnPalletInCVFwdJog;
_p3 := NOT gCtrl.main.noFaults;
_p4 := gCtrl.main.btnStop;
IF gCtrl.palletDispenser.hmiBtnPalletInCVRevJog OR gCtrl.palletDispenser.hmiBtnPalletInCVFwdJog OR NOT gCtrl.main.noFaults OR gCtrl.main.btnStop THEN
    gCtrl.palletDispenser.hmiBtnPalletInCVFwd := FALSE;
END_IF;
IF _p1 OR _p2 OR _p3 OR _p4 THEN gCtrl.palletDispenser.hmiBtnPalletInCVRev := FALSE; END_IF;
END_PROGRAM
```

### Program Logical/MachineControl/palletinfauto (IEC) - app pallete infeed dispenser auto logic

#### Cyclic.st
```iecst
PROGRAM _CYCLIC
	(* Insert code here *)
	gCtrl.palletDispenser.clawsOpenTmr();

	IF ((gCtrl.palletDispenser.dispenseState <> 0) AND (NOT gCtrl.main.noFaults)) THEN
		gCtrl.palletDispenser.dispenseState := 0;
	END_IF;

	CASE gCtrl.palletDispenser.dispenseState OF

		PLT_DISPENSE_ZERO :
			IF gCtrl.main.modeAuto THEN//wait here for auto mode
				gCtrl.palletDispenser.dispenseState := PLT_DISPENSE_INIT;
				gCtrl.palletDispenser.hmiBtnClawsLiftToTop := 1;
			END_IF;

		PLT_DISPENSE_INIT: //make sure to start at top
			IF gCtrl.palletDispenser.atTop THEN
				gCtrl.palletDispenser.hmiBtnPalletClawsOpenClose := 1;//CLOSE CLAWS
				gCtrl.palletDispenser.dispenseState := PLT_DISPENSE_IDLE;
				gCtrl.palletDispenser.dispenseDN := FALSE;
				gCtrl.palletDispenser.dispenseIP := FALSE;
				gCtrl.palletDispenser.dispenseReq := FALSE;
			END_IF;

		PLT_DISPENSE_IDLE:

			gCtrl.palletDispenser.dispenseDN := FALSE;
			gCtrl.palletDispenser.dispenseIP := FALSE;

			IF gCtrl.palletDispenser.dispenseReq THEN
				gCtrl.palletDispenser.dispenseIP := TRUE;
				gCtrl.palletDispenser.hmiBtnClawsLiftToBottom := 1;//GO TO BOTTOM
				gCtrl.palletDispenser.dispenseState := PLT_DISPENSE_TOBOTTOM;
			END_IF;

		PLT_DISPENSE_TOBOTTOM://wait to bottom
			IF gCtrl.palletDispenser.atBottom THEN//WAIT TO GET TO BOTTOM
				gCtrl.palletDispenser.hmiBtnPalletClawsOpenClose := 0;//OPEN CLAWS
				gCtrl.palletDispenser.clawsOpenTmr.IN := 0;
				gCtrl.palletDispenser.clawsOpenTmr.PT := T#3s;
				gCtrl.palletDispenser.dispenseState := PLT_DISPENSE_WTCLAWSOPN;
			END_IF;

		PLT_DISPENSE_WTCLAWSOPN://WAIT FOR CLAWS TO OPEN
			gCtrl.palletDispenser.clawsOpenTmr.IN := 1;
			IF gCtrl.palletDispenser.clawsOpenTmr.Q THEN
				gCtrl.palletDispenser.hmiBtnClawsLiftToMidLo := 1;//move to MID low
				gCtrl.palletDispenser.dispenseState := PLT_DISPENSE_TOMID;
			END_IF;

		PLT_DISPENSE_TOMID://WAIT FOR MID POSITION
			IF gCtrl.palletDispenser.atMidLo THEN//Wait for At mit Low
				gCtrl.palletDispenser.hmiBtnPalletClawsOpenClose := 1;//CLOSE CLAWS

				gCtrl.palletDispenser.clawsOpenTmr.IN := 0;
				gCtrl.palletDispenser.clawsOpenTmr.PT := T#3s;
				gCtrl.palletDispenser.dispenseState := PLT_DISPENSE_WTCLAWSCLS;
			END_IF;

		PLT_DISPENSE_WTCLAWSCLS://WAIT FOR CLAWS TO CLOSE
			gCtrl.palletDispenser.clawsOpenTmr.IN := 1;
			IF gCtrl.palletDispenser.clawsOpenTmr.Q THEN
				gCtrl.palletDispenser.hmiBtnClawsLiftToTop := 1;
				gCtrl.palletDispenser.dispenseState := PLT_DISPENSE_DN;
			END_IF;

		PLT_DISPENSE_DN://END OF DISPENSE CYCLE
			IF gCtrl.palletDispenser.atTop THEN
				gCtrl.palletDispenser.dispenseDN := TRUE;
				gCtrl.palletDispenser.dispenseReq := FALSE;
				gCtrl.palletDispenser.dispenseState := PLT_DISPENSE_IDLE;
			END_IF;

		ELSE

	END_CASE;

END_PROGRAM
```

### Program Logical/MachineControl/palletdischarge (IEC) - app pallet discharge conveyer

#### Cyclic.ld
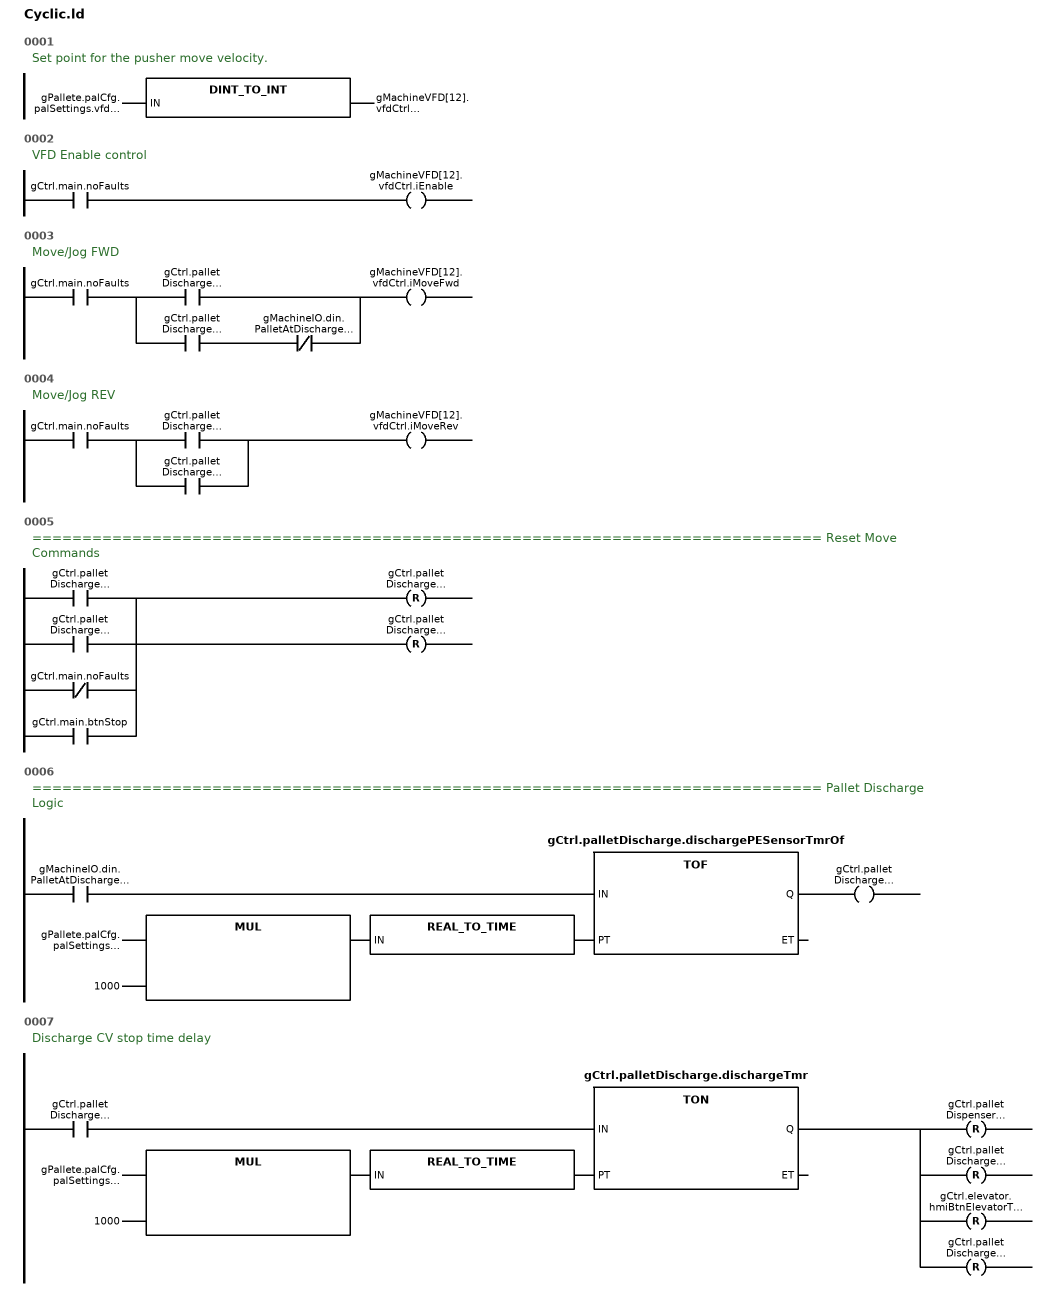
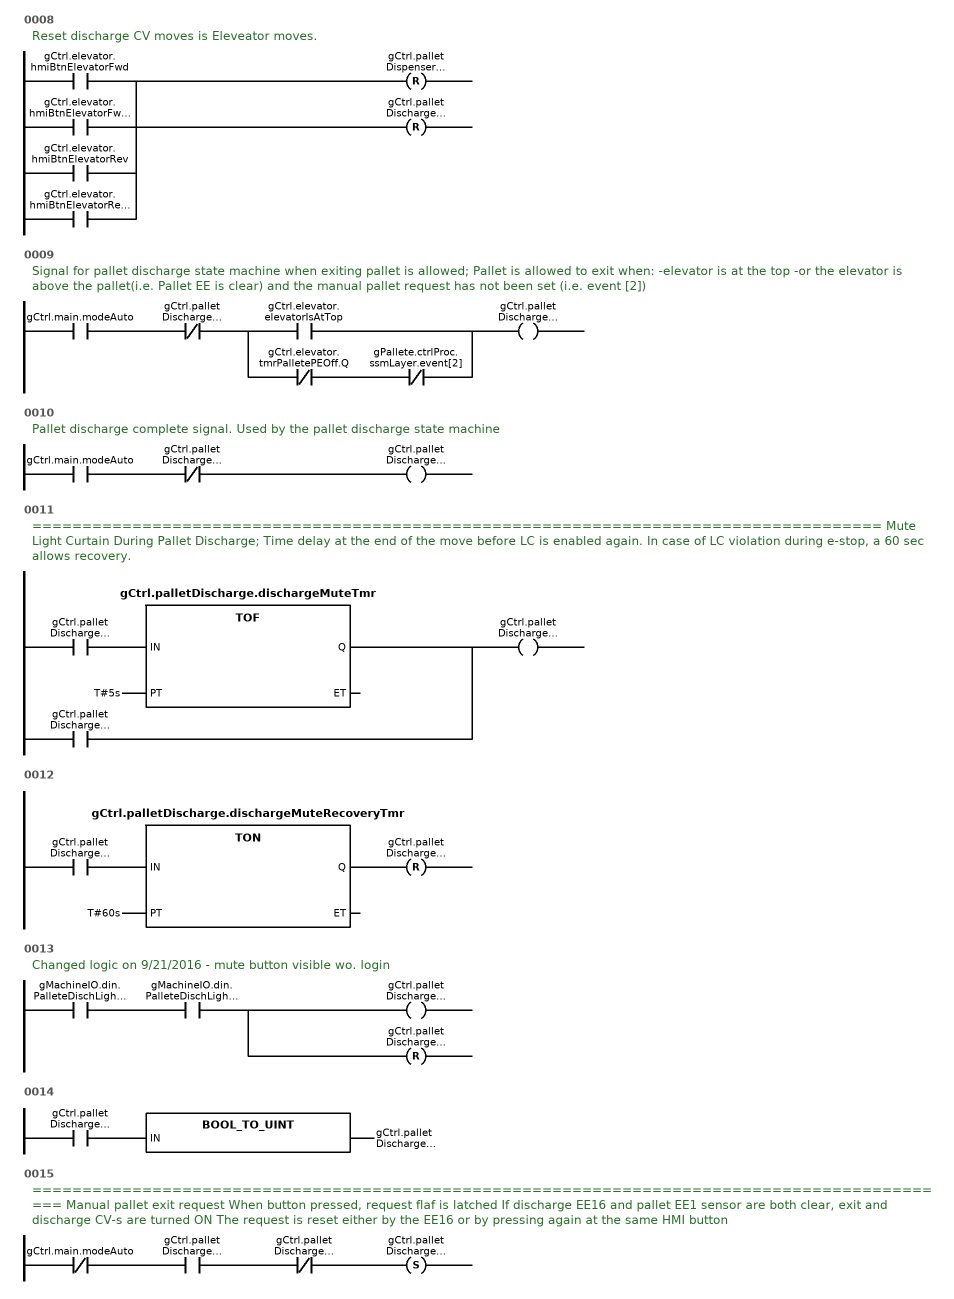
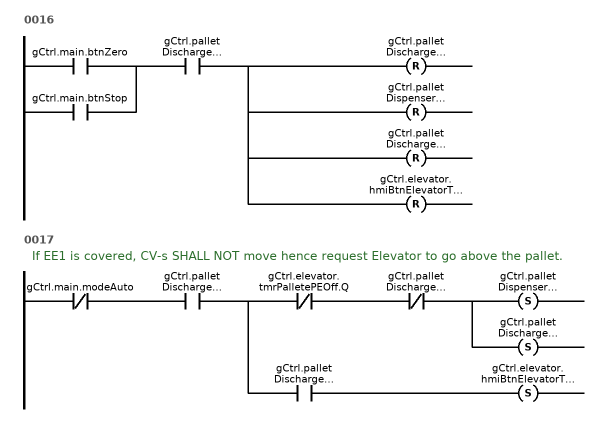
Ladder, written as Structured Text:
```iecst
PROGRAM _CYCLIC
VAR
    _p1 : BOOL;
    _p2 : BOOL;
    _p3 : BOOL;
    _p4 : BOOL;
    _p5 : BOOL;
    _p6 : BOOL;
    _p7 : BOOL;
    _p8 : BOOL;
    _p9 : BOOL;
    _p10 : BOOL;
    _p11 : BOOL;
    _p12 : BOOL;
    _p13 : BOOL;
    _p14 : BOOL;
END_VAR
(* Network 1: Set point for the pusher move velocity. *)
gMachineVFD[12].vfdCtrl.iVelocitySetPoint := DINT_TO_INT(gPallete.palCfg.palSettings.vfd[12].velocity_rpm);

(* Network 2: VFD Enable control *)
gMachineVFD[12].vfdCtrl.iEnable := gCtrl.main.noFaults;

(* Network 3: Move/Jog FWD *)
gMachineVFD[12].vfdCtrl.iMoveFwd := gCtrl.main.noFaults AND (gCtrl.palletDischarge.hmiBtnPalletDischargeCVFwd OR (gCtrl.palletDischarge.hmiBtnPalletDischargeCVFwdJog AND NOT gMachineIO.din.PalletAtDischarge_EE16));

(* Network 4: Move/Jog REV *)
gMachineVFD[12].vfdCtrl.iMoveRev := gCtrl.main.noFaults AND (gCtrl.palletDischarge.hmiBtnPalletDischargeCVRev OR gCtrl.palletDischarge.hmiBtnPalletDischargeCVRevJog);

(* Network 5: =============================================================================== Reset Move Commands *)
_p1 := gCtrl.palletDischarge.hmiBtnPalletDischargeCVRevJog;
_p2 := gCtrl.palletDischarge.hmiBtnPalletDischargeCVFwdJog;
_p3 := NOT gCtrl.main.noFaults;
_p4 := gCtrl.main.btnStop;
IF _p1 OR _p2 OR NOT gCtrl.main.noFaults OR gCtrl.main.btnStop THEN
    gCtrl.palletDischarge.hmiBtnPalletDischargeCVFwd := FALSE;
END_IF;
IF _p1 OR _p2 OR _p3 OR _p4 THEN gCtrl.palletDischarge.hmiBtnPalletDischargeCVRev := FALSE; END_IF;

(* Network 6: =============================================================================== Pallet Discharge Logic *)
gCtrl.palletDischarge.dischargePESensorTmrOf(IN := gMachineIO.din.PalletAtDischarge_EE16, PT := REAL_TO_TIME(gPallete.palCfg.palSettings.timers.EE16OfDebounce * 1000));
gCtrl.palletDischarge.dischargePESensor := gCtrl.palletDischarge.dischargePESensorTmrOf.Q;

(* Network 7: Discharge CV stop time delay *)
gCtrl.palletDischarge.dischargeTmr(IN := gCtrl.palletDischarge.dischargePESensor, PT := REAL_TO_TIME(gPallete.palCfg.palSettings.timers.onDlyPalleteDischargeEE16 * 1000));
_p5 := gCtrl.palletDischarge.dischargeTmr.Q;
IF gCtrl.palletDischarge.dischargeTmr.Q THEN gCtrl.palletDispenser.hmiBtnPalletInCVFwd := FALSE; END_IF;
IF _p5 THEN
    gCtrl.palletDischarge.hmiBtnPalletDischargeCVFwd := FALSE;
    gCtrl.elevator.hmiBtnElevatorToAbovePallete := FALSE;
    gCtrl.palletDischarge.palletManualExitRequest := FALSE;
END_IF;

(* Network 8: Reset discharge CV moves is Eleveator moves. *)
_p6 := gCtrl.elevator.hmiBtnElevatorFwd;
_p7 := gCtrl.elevator.hmiBtnElevatorFwdJog;
_p8 := gCtrl.elevator.hmiBtnElevatorRev;
_p9 := gCtrl.elevator.hmiBtnElevatorRevJog;
IF gCtrl.elevator.hmiBtnElevatorFwd OR gCtrl.elevator.hmiBtnElevatorFwdJog OR gCtrl.elevator.hmiBtnElevatorRev OR gCtrl.elevator.hmiBtnElevatorRevJog THEN
    gCtrl.palletDispenser.hmiBtnPalletInCVFwd := FALSE;
END_IF;
IF _p6 OR _p7 OR _p8 OR _p9 THEN gCtrl.palletDischarge.hmiBtnPalletDischargeCVFwd := FALSE; END_IF;

(* Network 9: Signal for pallet discharge state machine when exiting pallet is allowed; Pallet is allowed to exit when: -elevator is at the top -or the elevator is above the pallet(i.e. Pallet EE is clear) and the manual pallet request has not been set (i.e. event [2]) *)
_p10 := gCtrl.main.modeAuto AND NOT gCtrl.palletDischarge.dischargePESensor;
gCtrl.palletDischarge.isDischargeAllowed := _p10 AND (gCtrl.elevator.elevatorIsAtTop OR (NOT gCtrl.elevator.tmrPalletePEOff.Q AND NOT gPallete.ctrlProc.ssmLayer.event[2]));

(* Network 10: Pallet discharge complete signal. Used by the pallet discharge state machine *)
gCtrl.palletDischarge.dischargeDN := gCtrl.main.modeAuto AND NOT gCtrl.palletDischarge.hmiBtnPalletDischargeCVFwd;

(* Network 11: ===================================================================================== Mute Light Curtain During Pallet Discharge; Time delay at the end of the move before LC is enabled again. In case of LC violation during e-stop, a 60 sec allows recovery. *)
gCtrl.palletDischarge.dischargeMuteTmr(IN := gCtrl.palletDischarge.hmiBtnPalletDischargeCVFwd, PT := T#5s);
gCtrl.palletDischarge.muteLightCurtainDuringDischarge := gCtrl.palletDischarge.dischargeRecoveryIP OR gCtrl.palletDischarge.dischargeMuteTmr.Q;

(* Network 12 *)
gCtrl.palletDischarge.dischargeMuteRecoveryTmr(IN := gCtrl.palletDischarge.dischargeRecoveryIP, PT := T#60s);
IF gCtrl.palletDischarge.dischargeMuteRecoveryTmr.Q THEN
    gCtrl.palletDischarge.dischargeRecoveryIP := FALSE;
END_IF;

(* Network 13: Changed logic on 9/21/2016 - mute button visible wo. login  *)
_p11 := gMachineIO.din.PalleteDischLightCurtain_OSSD1 AND gMachineIO.din.PalleteDischLightCurtain_OSSD2;
gCtrl.palletDischarge.dischargeRecoveryVisible2 := _p11;
IF _p11 THEN gCtrl.palletDischarge.dischargeRecoveryIP := FALSE; END_IF;

(* Network 14 *)
gCtrl.palletDischarge.dischargeRecoveryVisible := BOOL_TO_UINT(gCtrl.palletDischarge.dischargeRecoveryVisible2);

(* Network 15: ============================================================================================= Manual pallet exit request When button pressed, request flaf is latched If discharge EE16 and pallet EE1 sensor are both clear, exit and discharge CV-s are turned ON The request is reset either by the EE16 or by pressing again at the same HMI button *)
IF NOT gCtrl.main.modeAuto AND gCtrl.palletDischarge.hmiBtnPalletManualExit AND NOT gCtrl.palletDischarge.palletManualExitRequest THEN
    gCtrl.palletDischarge.palletManualExitRequest := TRUE;
END_IF;

(* Network 16 *)
_p12 := (gCtrl.main.btnZero OR gCtrl.main.btnStop) AND gCtrl.palletDischarge.palletManualExitRequest;
IF _p12 THEN
    gCtrl.palletDischarge.palletManualExitRequest := FALSE;
    gCtrl.palletDispenser.hmiBtnPalletInCVFwd := FALSE;
    gCtrl.palletDischarge.hmiBtnPalletDischargeCVFwd := FALSE;
    gCtrl.elevator.hmiBtnElevatorToAbovePallete := FALSE;
END_IF;

(* Network 17: If EE1 is covered, CV-s SHALL NOT move hence request Elevator to go above the pallet. *)
_p13 := NOT gCtrl.main.modeAuto AND gCtrl.palletDischarge.palletManualExitRequest;
_p14 := _p13 AND NOT gCtrl.elevator.tmrPalletePEOff.Q AND NOT gCtrl.palletDischarge.dischargePESensor;
IF _p14 THEN
    gCtrl.palletDispenser.hmiBtnPalletInCVFwd := TRUE;
    gCtrl.palletDischarge.hmiBtnPalletDischargeCVFwd := TRUE;
END_IF;
IF _p13 AND gCtrl.palletDischarge.dischargePESensor THEN
    gCtrl.elevator.hmiBtnElevatorToAbovePallete := TRUE;
END_IF;
END_PROGRAM
```

### Program Logical/MachineControl/drycycle (IEC) - app dry cycle machine

#### Variables.var
```iecst
VAR
	elevatorTimer : TON := (0);
END_VAR
```

#### Cyclic.st
```iecst
PROGRAM _CYCLIC
	(* Insert code here *)
	elevatorTimer();

	IF ((dryCycleState <> 0) AND (NOT gCtrl.main.noFaults)) THEN
		dryCycleState := 0;
	END_IF;

	CASE dryCycleState OF
		0 : IF gCtrl.main.testBit1 THEN//wait here
				gCtrl.main.testBit1 := 0;
				dryCycleState := 1;
				elevatorTimer.IN := 0;
				elevatorTimer.PT := REAL_TO_UDINT(gPallete.palCfg.palSettings.timers.dlyTableLayerRdyToElevMove * 1000);
			END_IF;
		1: //wait a delay before start moving elevator
			elevatorTimer.IN := 1;
			IF elevatorTimer.Q THEN
				dryCycleState := 20;
				gCtrl.elevator.hmiBtnElevatorFwd := 1;//move elevator
				elevatorTimer.IN := 0;
				elevatorTimer.PT := REAL_TO_UDINT(gConfigApp.options.tmDryCycleElevatorUp * 1000) * gCtrlAnimation.currentLayer + REAL_TO_UDINT(gConfigApp.options.tmDryCycleLayerZeroOffset * 1000);
			END_IF;

		20://box pusher is done
			elevatorTimer.IN := 1;
			IF elevatorTimer.Q THEN
				elevatorTimer.IN := 0;
				gCtrl.elevator.hmiBtnElevatorFwd := 0;
				gCtrl.transfertable.hmiBtnTableFwd := 1;
				dryCycleState := 30;
			END_IF;
		30:
			IF gCtrl.transfertable.isTableAtPallete THEN
				gCtrl.squaring.hmiBtnSidePlatesExtRet := 1;
				gCtrl.retainerbar.hmiBtnRetainterBarFwd := 1;

				elevatorTimer.IN := 1;
				elevatorTimer.PT := T#3s;

				dryCycleState := 35;
			END_IF;
		35:
			IF elevatorTimer.Q THEN
				gCtrl.transfertable.hmiBtnTableRev := 1;
				dryCycleState := 40;
			END_IF;

		40://
			IF gCtrl.transfertable.isTableAtGrouping THEN
				gCtrl.squaring.hmiBtnSidePlatesExtRet := 0;
				gCtrl.retainerbar.hmiBtnRetainterBarRev := 1;
				gCtrl.elevator.hmiBtnElevatorToGrouping := 1;
				dryCycleState := 50;
			END_IF;
		50://wait for elevator to come back home
			IF gCtrl.elevator.elevatorIsAtHome THEN
				dryCycleState := 0;
				gCtrl.main.testBit3 := 1;
			END_IF;
		60://dry cycle is done

		ELSE

	END_CASE;

END_PROGRAM
```

### Program Logical/MachineControl/drycypal (IEC) - app dry pallete

#### Variables.var
```iecst
VAR
	palleteTimer : TON := (0);
END_VAR
```

### Package Logical/Simulation - application simulation and testing tasks and logic

### Program Logical/Simulation/counter

#### counter.c
```c
/********************************************************************
 * COPYRIGHT -- HP
 ********************************************************************
 * Program: counter
 * File: counter.c
 * Author: goran
 * Created: March 07, 2013
 ********************************************************************
 * Implementation of program counter
 ********************************************************************/

#include <bur/plctypes.h>

#ifdef _DEFAULT_INCLUDES
	#include <AsDefault.h>
#endif

_LOCAL int counter;

void _INIT counterINIT(void)
{
	/* TODO: Add code here */
}

void _CYCLIC counterCYCLIC(void)
{
	/* TODO: Add code here */
	counter++;
	counter++;

}
```

### Program Logical/Simulation/IOsim (ANSIC)

#### IOsim.c - Cyclic code
```c
/********************************************************************
 * COPYRIGHT -- Gainco
 ********************************************************************
 * Program: IO
 * File: IO.c
 * Author: DavidT
 * Created: July 13, 2010
 ********************************************************************
 * Implementation of program IO
 ********************************************************************/

#include <bur/plctypes.h>

#ifdef _DEFAULT_INCLUDES
#include <AsDefault.h>
#endif

#include <..\globalvar.h>
#include <..\..\GlobalDef.h>
#include <..\..\GlobalDecl.h>
//#include "..\\..\\RecFIFO\\fifotest\\fifoif.h"
#include "..\\..\\bglib\\bgsprintf.h"
#include "..\\..\\bglib\\bgsprintf.c"

_LOCAL  BOOL   _inZeroSensor; //n-1 value
_LOCAL  BOOL   _inBeltFlite;  //n-1 value

/*
###############################################################################
Utilities
###############################################################################
*/

/**
 Simple logging
 Log goes to an array of PV strings > see _LOCAL STRING log[][] variable below
 Log output is visible via Automation Studio watch window
 Example of a log statement used within the code is:
 DBG(lgr, "This is log example. %d ", value1);
 To complety disable logging from this source file, change next line to: #if 0
IMPORTANT:
==========
DBGINIT() statement MUST BE PLACED as a first statement within the task _INIT function!
Example:
void _INIT myTaskINIT(void)
{
	//TODO: Add code here
	//init logger object
	DBGINIT(lgr, log, LOG_ENTRY_COUNT, LOG_ENTRY_LENGTH);
}
*/
#if 1
#include <../../bglib/bgPVLogger.c>
#define LOG_ENTRY_COUNT 20	//max number of log entries
#define LOG_ENTRY_LENGTH  32 //max length of individual log message. Longer msg are truncated
_LOCAL STRING log[LOG_ENTRY_COUNT][LOG_ENTRY_LENGTH]; //log output visible from Automation Studio!
static bgPVLogger_typ lgr;	//PV logger object
#else
#define DBG(loggerInstance, format, args...) ;
#define DBGINIT(loggerInstance, logoutput, logEntryCount, logEntrySize)  ;
#endif

#define TK_CYCLE_TIME_Xms 0.01
#define TK_CYCLE_TIME_counts 10
//stage hopper gate control functions for all hoppers
static void stageHoppersGatesClose()
{
	int i;
	for (i=0; i<Config.Cfg_NumTakeoffs; i++)
	{
		Stage[i] = 1;//1 (energized) keeps the gates closed
	}
}

static void stageHoppersGatesOpen()
{
	int i;
	for (i=0; i<Config.Cfg_NumTakeoffs; i++)
	{
		Stage[i] = 0; //0 (not energized) keeps the gates open
	}
}

static BOOL isQCRequiredCurrentStation()
{
	if (QCbypass[OutfeedStation-1] || ((qc[0].QCLoginedIn == 0) && (qc[1].QCLoginedIn == 0)) )
		return 0;//not required when: not request by the HMI and both QC station are not logged in

	return 1;
}

//Find if QC required for the pocket that's going to be dropped next into the outfeed hopper
//OutfeedStation contains number (i.e. 1..16) of the outfeed station that's currently beeing
//dumped into the outfeed hopper (note that it starts with 1 not with 0!)
//
static BOOL isQCRequiredNextStation()
{
int outfeedStationIndexCurrent;
int outfeedStationIndexNext;

	//if OutfeedStation == 0 > no dumping into the outfeed, we are in the search for
	//zero tab > nothing to do
	if(!OutfeedStation)
		return 0;

	//find index (0 based) of the station beeing dumped into the outfeed hopper
	outfeedStationIndexCurrent = OutfeedStation - 1;

	//check if station that's comming next shall be QC-ed
	if(outfeedStationIndexCurrent){
		outfeedStationIndexNext = outfeedStationIndexCurrent - 1;
		if (QCbypass[outfeedStationIndexNext] || (qc[0].QCLoginedIn == 0) )
			return 0;
	}

	//note that for the last station (i.e. OutfeedStation==1), the next station # is Config.Cfg_NumTakeoffs
	if(!outfeedStationIndexCurrent){
		outfeedStationIndexNext = Config.Cfg_NumTakeoffs - 1;
		if (QCbypass[outfeedStationIndexNext] || (qc[0].QCLoginedIn == 0) )
			return 0;
	}

	return 1;
}

//q - qc station index (0 or 1)
static BOOL isQCInspectionActive(int q)
{
	//check if QC inspection is active
	if (qc[q].QCStarted && qc[q].QCLoginedIn)
		return 1;

	return 0;
}

static BOOL isQCLogged_NotStarted(int q)
{
	//check if QC inspection is active
	if (!qc[q].QCStarted && qc[q].QCLoginedIn)
		return 1;

	return 0;
}

//Advance outfeed to the next station
static void outfeedAdvance()
{
	QCselect[0] = 0;
	QCselect[1] = 0;
	if (OutfeedStation == 1)
	{
		ZeroFlag = 0;
		OutfeedStation = 0;
		outstate = 12;
	}
	else
	{
		BeltClutch = 1;
		OutfeedStation--;
		outstate++;
	}

}

//Detect if stopping/pausing outfeed is allowed
static BOOL isOutfeedPauseBlocked()
{
	//Don't allow stop (pause) outfeed SM while belt clutch is on during product indexing
	//That way, we'll avoid a problem with partial dumping of the bin/station content (i.e. if
	//indexing stopped when some product dropped and some product remains in the pocket)
	if( (outstate >= 9) && (outstate <= 11) && BeltClutch )
		return 1; //if above states are active and the belt clutch is on > that's indexing. Don't allow STOP to take place

	//Don't allow stop/pause when the first pocket to be dropped is about to reach the desitnation
	//state 8 is active afer product is dropped onto the belt, until the lead pocket gets dropped into the outfeed hopper
	if( (outstate == 8) && (ZtoDump >= FlightCounter))
		return 1;

	return 0;
}

//Process MasterMode signal and control outfeed state machine
//based upon MasterMode changes
static BOOL outfeedMasterModeLogic()
{
static BOOL _BeltClutch;
static DINT _pauseOperation;
int   i,j;

	//process MasterMode changes
	if (MasterMode != _MasterMode)
	{
		//Previos mode
		switch (_MasterMode)
		{
			case RUN_MODE:
				_BeltClutch = BeltClutch;//preserve belt clutch state when leaving RUN mode
			break;
		}

		//New mode
		switch (MasterMode)
		{
			case STOP_MODE:
				//check if stop/pause is allowed
				if( isOutfeedPauseBlocked() ){
					//pause is blocked, can't switch to stopped mode! wait here until it gets unblocked (i.e. belt turns off)
					//when exiting here, _MasterMode does not get updated. As a result, we'll keep
					//comming back to this point until pause gets unblocked
					return 0;//make sure outfeed SM continues execution!!!
				}

				//entering STOP mode from any other state
				//_BeltClutch = BeltClutch;//preserve belt clutch state
				BeltClutch  = 0;//stop belt
				//NOTE: SM stops executing in this mode, see below
			break;

			case RUN_MODE:
				BeltClutch = _BeltClutch;//restore belt clutch state (preserved when exited RUN state)
				ZeroFlag = 0;//make sure to clear this flag before restoring RUN state

				//when starting RUN from states:
				//0-stopped
				//1-filling
				//3- washdown
				//force the outstate to start at first step in the RUN state (2)
				if(outstate <= 3){
					outstate = 2;
				}else{
					//BAND AID TO MAKE SURE OUTFEED BELT MOVES WHEN SWITCHING TO RUN STATE
					switch(outstate){
						case 5:
						case 6:
						case 8:
						case 9:
						case 11:
							if(!BeltClutch){
								DBG(lgr, "beltOFF,ONreq! otst=%d", outstate);
								BeltClutch = 1;
							}
						break;
					}
				}

				//VERY DIFFICULT PROBLEM DISCOVERED AT MILFORD
				if(outstate == 10){
					OutfeedDumped = 1;//restart handshake to a point that the hopper can pick it up without locking up
				}

				//otherwise, don't touch outstate > it will continue execution from the point where it stopped (outstate > 3)
			break;

			case FILL_MODE:
//				outstate = 1; //start fill
				//check if stop/pause is allowed
				if( isOutfeedPauseBlocked() ){
					//pause is blocked, can't switch to stopped mode! wait here until it gets unblocked (i.e. belt turns off)
					//when exiting here, _MasterMode does not get updated. As a result, we'll keep
					//comming back to this point until pause gets unblocked
					return 0;//make sure outfeed SM continues execution!!!
				}

				//entering STOP mode from any other state
				//_BeltClutch = BeltClutch;//preserve belt clutch state
				BeltClutch  = 0;//stop belt
				//NOTE: SM stops executing in this mode, see below

				//case 1: // fill
					BeltClutch  = 0;
					QCselect[0] = 0;
					QCselect[1] = 0;
					stageHoppersGatesClose();
				//break;

			break;

			case WASHDOWN_MODE:
				outstate = 3; // goto washdown
			break;
		}

		DBG(lgr, "outfeed MasterMode=%d", MasterMode);
		_MasterMode = MasterMode;
	}

	//pause request set
	if(gUdpCmdMsg.outfeed.pauseOperation && !_pauseOperation){
		//same as stop mode
		if(MasterMode == RUN_MODE){

			//check if stop/pause is allowed
			if( isOutfeedPauseBlocked() ){
				//pause is blocked! wait here until it gets unblocked (i.e. belt turns off)
				//when exiting here, _pauseOperation does not get updated. As a result, we'll keep
				//comming back to this point until pause gets unblocked
				return 0;//make sure outfeed SM continues execution!!!
			}

			//pause feature is supported only in RUN mode
			_BeltClutch = BeltClutch;//preserve belt clutch state
			BeltClutch  = 0;//stop belt
		}
		_pauseOperation = gUdpCmdMsg.outfeed.pauseOperation;
	}

	//pause request reset
	if(!gUdpCmdMsg.outfeed.pauseOperation && _pauseOperation){
		if(MasterMode == RUN_MODE){
			//pause feature is supported only in RUN mode
			BeltClutch = _BeltClutch;//restore belt clutch state
			_pauseOperation = gUdpCmdMsg.outfeed.pauseOperation;
		}
	}

	//if STOP mode active > exit here (i.e. don't execute SM)
	if((MasterMode == STOP_MODE) || (MasterMode == FILL_MODE) || (  (MasterMode == RUN_MODE) && _pauseOperation) ){
		return 1;//returning 1 means that outfeed SM will not be executed!!!
	}

	return 0;
}

_LOCAL BOOL lastSelectedQC;

//outfeed state machine
void outfeed(void)
{
int   i,j;
static DINT _OutfeedDumped;

	//process MasterMode and control outfeed SM (outstate)
	//if outfeed SM should be stopped (i.e. not executed, the function returns 1)
	if(outfeedMasterModeLogic()){
		return;
	}

	//log outstate change
	if(outstate != _outstate)
	{
		_outstate = outstate;
		DBG(lgr, "outfeed sm: %d", outstate);
	}

	//log OutfeedDumped change
	if(OutfeedDumped != _OutfeedDumped)
	{
		_OutfeedDumped = OutfeedDumped;
		DBG(lgr, "OfD=%d, Qsl=%d, Qst=%d OfHD=%d", OutfeedDumped, QCselect[0], qc[0].QCStarted, Weigh[1]);

		bgsprintf(gDiagEventRecToFIFO.eventText, "OfD=%d, Qsl=%d, Qst=%d OfHD=%d", OutfeedDumped, QCselect[0], qc[0].QCStarted, Weigh[1]);
		gDiagEventRecToFIFO.eventId = 103;
		captureDiagEvent(gDiagEventRecToFIFO.eventId, gDiagEventRecToFIFO.eventText);
	}

	//outfeed state machine (SM)
	switch (outstate)
	{
	case 0: //stop
		BeltClutch  = 0;
		QCselect[0] = 0;
		QCselect[1] = 0;
		stageHoppersGatesClose();
	break;

	case 1: // fill
		BeltClutch  = 0;
		QCselect[0] = 0;
		QCselect[1] = 0;
		stageHoppersGatesClose();
	break;

	case 2: // run
		//set hw for run
		BeltClutch  = 0;
		QCselect[0] = 0;
		QCselect[1] = 0;
		stageHoppersGatesClose();
		outstate = 4;
	break;

	case 3: // washdown
		// set i/o for washdown
		BeltClutch  = 1;
		QCselect[0] = 0;
		QCselect[1] = 0;
		stageHoppersGatesOpen();
	break;

	case 4: // start outfeed
		BeltClutch = 1;
		outstate++;
	break;

	case 5:  // look for zero tab
		if (ZeroFlag)
		{
			ZeroFlag = 0;
			stop1dly = 0.0;
			outstate++;
		}
	break;

	case 6:  // stop 1 delay after zero tab detected
		stop1dly += .001;
		if (stop1dly > Config.Cfg_Stop1dly)
		{
			BeltClutch = 0;
			ZtoDump = 0;
			Stagedly1 = 0.0;
			Stagedly2 = 0.0;
			stageHoppersGatesOpen();//as soon as the belt stops, dump product onto the outfeed belt
			outstate++;
		}
	break;

	case 7:  // Delay for Dumping Staging Hoppers & dump to outfeed belt

		Stagedly1 += TK_CYCLE_TIME_Xms;
		if (Stagedly1 >= gUdpCmdMsg.outfeed.stagingHopperOpenDuration)
		{
			stageHoppersGatesClose();
//			stageHoppersGatesOpen();

			Stagedly2 += TK_CYCLE_TIME_Xms;
			if (Stagedly2 >= gUdpCmdMsg.outfeed.outfeedBeltCycleStartDelay)
			{
				FltCntFlg  = 0;//reset flight counter
				//stageHoppersGatesClose();
				BeltClutch = 1; // Start Moving belt
				outstate++;
			}
		}
	break;

	case 8:  // Zero to first Dump
		if (FltCntFlg)
		{
			FltCntFlg = 0;
			ZtoDump++;
			if (ZtoDump > FlightCounter)
			{
				stop2dly = 0.0;
				OutfeedStation = Config.Cfg_NumTakeoffs;//set the station that will be processed first at the outfeed hopper
				outstate++;
			}
		}
	break;

	case 9:  // Stop 2 DLY, delay after a flight that contains product that shall be dropped first is detected
		stop2dly += TK_CYCLE_TIME_Xms;
		if (stop2dly > Config.Cfg_Stop2dly)
		{
			BeltClutch = 0;//stop the outfeed belt
			OutfeedDumped = 1;//request to outfeed hopper to weigh the product
			QCskip = 0;//QC skip is cleared (i.e. QC shall be executed if possible/required)
			outstate++;
		}
	break;

	case 10:  // startup belt
	/*
	IMPORTANT: in this state, a handshake between this SM and the outfeed hopper SM takes place
	For outfeed hopper see master.c, outfeed() function, state APP4_DUMP and function call:
	HopperOutfeedDump(Ch)

	Chain of events:

	outfeedSM, state 9:
	OutfeedDumped = 1 //request to hopper SM to weigh product

	outfeedHopperSM, state APP4_FILL:
	if(	OutfeedDumped == 1)
	goto NextStep //i.e. measure product dumpped into the outfeed hopper

	outfeedHopperSM, state APP4_DUMP:
	if( CaptureWeight is GoodForQC)
	OutfeedDumped = 2 //signal to outfeed SM that product weight is GOOD
	else
	OutfeedDumped = 5 //signal to outfeed SM that product weight is NO GOOD
	etc.
	*/
		switch(OutfeedDumped){
		case 0:	//Outfeed hopper is done. Product is dropped!
			//Continue here and decide if QC shall be started for this product

			if(QCskip || !isQCRequiredCurrentStation()){
				//QCskip == 1 when product weight is NO GOOD (small weight) for QC
				//QC not required > advance outfeed conveyer to the next station
				outfeedAdvance(); //outfeed SM will be changed within this call!
				return;
			}

			//Check if current product shall be QC-ed AND the product is dumpped at the QC
			if( isQCRequiredCurrentStation() && isQCLogged_NotStarted(0) && (QCselect[0] == 1) ){
				//Yes, current product shall be QC-ed AND the product is dumpped at the QC (QC deverter gate is towards QC)
				qc[0].OutfeedRecId = getOutfeedRecId();
				qc[0].QCcurStation = OutfeedStation;
				qc[0].QCStarted   = 1;
				qc[0].QCtotaltime = 0.0;
			}else
			if( isQCRequiredCurrentStation() && isQCLogged_NotStarted(1) && (QCselect[1] == 1) ){
				//Yes, current product shall be QC-ed AND the product is dumpped at the QC (QC deverter gate is towards QC)
				qc[1].OutfeedRecId = getOutfeedRecId();
				qc[1].QCcurStation = OutfeedStation;
				qc[1].QCStarted   = 1;
				qc[1].QCtotaltime = 0.0;
			}

			outfeedAdvance();
		break;
		case 1://set by outfeed sm (above) after product dumped into outfeed hopper for weighing
			//nothing to do > wait for outfeed hopper sm to change the state variable OutfeedDumped
			stop2dly = 0.0;
		break;
		case 2://set by the outfeed hopper sm after sufficent product weight detected at the outfeed scale

			if( !isQCRequiredCurrentStation() ){
			//QC is not required for the current station
			//not required when: no request by the HMI OR both QC station are NOT logged in
				QCselect[0] = 0;
				QCselect[1] = 0;

				stop2dly += TK_CYCLE_TIME_Xms;//wait for timer to expire before letting hopper sm to proceed
				if (stop2dly > 0.05){
					OutfeedDumped = 3;
				}
				return;
			}

			//YES, QC is required for the current station!

			if( isQCLogged_NotStarted(0) && isQCLogged_NotStarted(1) ){
				//Both are available for inspection

				//Select the QC that is different then the last one
				if(lastSelectedQC){
					QCselect[0] = 1;
					QCselect[1] = 0;
					qc[0].QCweight = App[1].Hopper.GrossWeight;
					lastSelectedQC = 0;
				}else{
					QCselect[0] = 0;
					QCselect[1] = 1;
					qc[1].QCweight = App[1].Hopper.GrossWeight;
					lastSelectedQC = 1;
				}
			}else
			if(isQCLogged_NotStarted(0)){
				//QC 0 is available for inspection

				QCselect[0] = 1;
				QCselect[1] = 0;
				qc[0].QCweight = App[1].Hopper.GrossWeight;
				lastSelectedQC = 0;
			}else
			if(isQCLogged_NotStarted(1)){
				//QC 1 is available for inspection

				QCselect[0] = 0;
				QCselect[1] = 1;
				qc[1].QCweight = App[1].Hopper.GrossWeight;
				lastSelectedQC = 1;
			}else{
				//no QC is available

				QCselect[0] = 0;
				QCselect[1] = 0;

				//check the qc mode
				if(qc[0].QCmode == 0){
					//QC mode is MUST DO QC > stop the outfeed until a QC is available (wait here)
					return;
				}
				//otherwise, advance the outfeed following a delay below
			}

			stop2dly += TK_CYCLE_TIME_Xms;//wait for timer to expire before letting hopper sm to proceed
			if (stop2dly > 0.65){//7/10/13 - increade delay to make sure that QC shoot moves to a position before weigh door gets opened
				OutfeedDumped = 3;
			}

	break;
	case 3:
	case 4:
	case 5:
	//nothing to do > wait for outfeed hopper sm to change the state variable OutfeedDumped
	break;
	}

	break;

	case 11:  // next flt
		if (FltCntFlg)
		{
			FltCntFlg = 0;
			stop2dly = 0.0;
			outstate = 9;
		}
	break;

	case 12:  // look for next zero
		BeltClutch = 1;
		outstate = 5;
	break;
	}

}

//Functions to support DO-s forcing from the host
static BOOL diagIsForceDOsActive()
{
	if( !gUdpCmdMsg.diag.io.enableDOForce ){
		return 0;
	}

	if( MasterMode != STOP_MODE ){
		return 0;
	}

	return 1;
}
static void diagForceDOs()
{
	int ii;

	if( !diagIsForceDOsActive() )
		return;

	//Following DO-s are controlled from this task
	//When DO force gets activagted, these DO-s are congtrolled directly by the host via UDP cmd msg
	BeltClutch = (gUdpCmdMsg.diag.io.outfeed.DOModule & 0x02) ? 1 : 0;
	QCselect[0] = (gUdpCmdMsg.diag.io.outfeed.DOModule & 0x10) ? 1 : 0;
	QCselect[1] = (gUdpCmdMsg.diag.io.outfeed.DOModule & 0x80) ? 1 : 0;

	for(ii=0; ii<YP_MAX_STATIONMODULES; ii++){
		Stage[ii*4 + 0] = (gUdpCmdMsg.diag.io.stations[ii].DOModule & 0x02) ? 1 : 0;
		Stage[ii*4 + 1] = (gUdpCmdMsg.diag.io.stations[ii].DOModule & 0x08) ? 1 : 0;
		Stage[ii*4 + 2] = (gUdpCmdMsg.diag.io.stations[ii].DOModule & 0x20) ? 1 : 0;
		Stage[ii*4 + 3] = (gUdpCmdMsg.diag.io.stations[ii].DOModule & 0x80) ? 1 : 0;
	}
}

//Process and detect belt zero signal rising edge
static void ioBeltZeroDetect()
{
	if (inBeltZero && !_inZeroSensor)  //Rising Edge
	{
		ZeroCount++;
		ZeroFlag = 1;
	}
	_inZeroSensor = inBeltZero;
}

//Flite sensor operation
//This function processes the flite sensor digital input
//During normal operation, flite sensor detects passing of each flite on the outfeed
//belt conveyer. Detecting flites is critical for the proper operation of the machine.
//In case of a flite sensor mulfunction (or erronius flite detection), machine operation
//may be severly disturbed.
//As a result, and in addition to the normal operation, this function provides
//funcionality to detect, report and handle common flite sensor errors
static void ioFliteDetectEx(ioFliteSensorDetector_typ* p)
{

	//single shot (cycle) flag
	p->oFliteSignalDetected = 0;

	switch(p->prvState){
		case 0: //at startup, init variables
			p->prvOnCounter = 0;
			p->prvOffCounter = 0;
			p->oPulseOffTimeMin = 1000;
			p->oPulseOffTimeMax = 0;
			p->oPulseOnTimeMin = 1000;
			p->oPulseOnTimeMax = 0;
			p->prvState = 5;
		break;
		case 5:	//belt off
		//when belt if off, flites are not moving, nothing to do

			if(!p->iBelt){
				p->oAlarmPulsOff = 0;
				p->oAlarmPulsOn = 0;
				p->oFliteSignalDetected = 0;
				p->oFliteCounter = 0;
				return;
			}

			//belt got turned on
			p->prvOffCounter = 0;
			p->prvOnCounter = 0;

			//depending on the current state of the flite sensor input
			//goto an appropirate state
			if(p->iFliteSensor){
				p->prvState = 20;//goto physical flite signal on
			}else{
				p->prvState = 10;//goto physical flite signal off
			}
		break;
		case 10://physical flite signal is off
			p->prvOffCounter += TK_CYCLE_TIME_counts; //measure the time in this state

			if(!p->iBelt){
				p->prvState = 5;//if belt turned off > goto belt off state
				return;
			}

			//pulse off duration too long?
			if(p->prvOffCounter > p->iPulseOffTimeMax){
				//trouble! sensor signal is off longer than expected!
				p->oAlarmPulsOff = 1;//generate alarm
				p->oFliteSignalDetected = 1;//create a fake flite signal detected indication (used by the machine logic)
				p->prvOnCounter = 0;//reset pulse on counter for the fake on signal generation
				p->prvState = 11;//pulse off is too long > simulate pulse on!
				return;
			}

			if(p->iFliteSensor){
				//ok, this is normal! pulse turned on
				//capture min/max off times
				if(p->prvOffCounter > p->oPulseOffTimeMax){
					p->oPulseOffTimeMax = p->prvOffCounter;
				}
				if(p->prvOffCounter < p->oPulseOffTimeMin){
					p->oPulseOffTimeMin = p->prvOffCounter;
				}

				p->oFliteSignalDetected = 1;//create a flite signal detected indication (used by the machine logic)
				p->prvOnCounter = 0;
				p->prvState = 15;//physical signal on filter
			}
		break;
		case 11://pulse off too long > simulate on pulse
			p->prvOnCounter+=TK_CYCLE_TIME_counts;

			if(!p->iBelt){
				p->prvState = 5;//if belt turned off > goto belt off state
				return;
			}

			if(p->iFliteSensor){
				p->prvState = 15;//ups! physical signal is on > good!
				p->prvOnCounter = 0;
				return;
			}

			//virtual on signal expired?
			if(p->prvOnCounter > p->iPulseOnTimeMax){
				p->prvOffCounter=0;
				p->prvState = 10;//back to physical pulse off
			}
		break;
		case 15://physical pulse on filter
			p->prvOnCounter+=TK_CYCLE_TIME_counts;

			if(!p->iBelt){
				p->prvState = 5;//goto belt off
				return;
			}

			if(p->prvOnCounter > p->iPulseOnFilterTime){
				//on filter! disable any processing for the specified interval
				p->prvState = 20;//physical signal on
				return;
			}
		break;
		case 20://physical signal is on
			p->prvOnCounter+=TK_CYCLE_TIME_counts;

			if(!p->iBelt){
				p->prvState = 5;//goto belt off
				return;
			}

			//pulse on duration too long?
			if(p->prvOnCounter > p->iPulseOnTimeMax){
				p->prvOffCounter = 0;
				p->oAlarmPulsOn = 1;//generate alarm
				p->prvState = 21;//signal on too long!
				return;
			}

			if(!p->iFliteSensor){
				//ok, this is normal! sensor signal turned off
				//capture min/max on times
				if(p->prvOnCounter > p->oPulseOnTimeMax){
					p->oPulseOnTimeMax = p->prvOnCounter;
				}
				if(p->prvOnCounter < p->oPulseOnTimeMin){
					p->oPulseOnTimeMin = p->prvOnCounter;
				}

				p->prvState = 10;//physical pulse off
				p->prvOffCounter = 0;
			}
		break;
		case 21://signal on too long > simulate off signal
			p->prvOffCounter+=TK_CYCLE_TIME_counts;

			if(!p->iBelt){
				p->prvState = 5;//goto belt off
				return;
			}

			if(!p->iFliteSensor){
				p->prvState = 10;//physical signal off
				p->prvOffCounter = 0;
				return;
			}

			//virtual signal off expired?
			if(p->prvOffCounter > p->iPulseOffTimeMax){
				p->prvOnCounter=0;
				p->oFliteSignalDetected = 1;//fake sensor signal
				p->prvState = 20;//back to physical pulse on
			}
		break;
	}
}

//Process and detect flight sensor signal
static void ioFliteDetect()
{
//#if 0
	ioFliteSensor.iBelt = BeltClutch;
	ioFliteSensor.iFliteSensor = inBeltFlite;
	ioFliteSensor.iPulseOnFilterTime = gUdpCmdMsg.outfeed.flightFilterCount;
	ioFliteSensor.iPulseOffTimeMax = (UDINT)(gUdpCmdMsg.outfeed.flightTimeMax * 1000.0);
	ioFliteSensor.iPulseOnTimeMax = (UDINT)(gUdpCmdMsg.outfeed.flightTimeMin * 1000.0);
	ioFliteDetectEx(&ioFliteSensor);

	if(ioFliteSensor.oAlarmPulsOff){
		ioFliteSensor.oAlarmPulsOff = 0;
		memset(gDiagEventRecToFIFO.eventText, 0, sizeof(gDiagEventRecToFIFO.eventText));
		bgsprintf(gDiagEventRecToFIFO.eventText, "flite signal OFF error (maxOffTime=%d[ms]", (UDINT)(ioFliteSensor.iPulseOffTimeMax));
		gDiagEventRecToFIFO.eventId = 101;
		captureDiagEvent(gDiagEventRecToFIFO.eventId, gDiagEventRecToFIFO.eventText);
	}

	if(ioFliteSensor.oAlarmPulsOn){
		ioFliteSensor.oAlarmPulsOn = 0;
		memset(gDiagEventRecToFIFO.eventText, 0, sizeof(gDiagEventRecToFIFO.eventText));
		bgsprintf(gDiagEventRecToFIFO.eventText, "flite signal ON error (maxOnTime=%d[ms]", (UDINT)(ioFliteSensor.iPulseOnTimeMax));
		gDiagEventRecToFIFO.eventId = 102;
		captureDiagEvent(gDiagEventRecToFIFO.eventId, gDiagEventRecToFIFO.eventText);
	}

	FltCntFlg = ioFliteSensor.oFliteSignalDetected;

//#endif

#if 0
	if (FltFilter == 0)
	{
		if (inBeltFlite && !_inBeltFlite)  //Rising Edge
		{
			FltCount++;
			FltFilter  = 1;
			FltCntFlg  = 1;
		}
	}
	else
	{
		FltFilter++;
		if (FltFilter>FltFilterCount)
		{
			FltFilter = 0;
		}
	}
	_inBeltFlite = inBeltFlite;
#endif
}

//generate delay timers using 1ms cycle time
static void	hopperDelayTimers()
{
	int i,j;

	for(i=0; i<DELAY_MAX; i++)
	{
		for(j=0; j<Config.Cfg_NumHoppers; j++)
		{
			if (IODelaySec[i][j] != -0.5)
			{
				if (IODelaySec[i][j] >= 0.0)
				{
					IODelaySec[i][j] -= TK_CYCLE_TIME_Xms;
					if (IODelaySec[i][j] < 0.0)
					{
						if (i == DELAY_LINE)
						{
							Line[j] = IODelayBit[DELAY_LINE][j];
						}
						else if (i == DELAY_WEIGH)
						{
							Weigh[j] = IODelayBit[DELAY_WEIGH][j];
						}
						else if (i == DELAY_BUFFER)
						{
							Buffer[j] = IODelayBit[DELAY_BUFFER][j];
						}
						else if (i == DELAY_1)
						{
							Delay1[j] = IODelayBit[DELAY_1][j];
						}
						IODelaySec[i][j] = -0.5;
					}
				}
			}
		}
	}
}
/*
###############################################################################
Task execution entry points: Init & Cyclic Functions
###############################################################################
*/
_INIT void DataINIT(void)
{
	int i, j;

	//init logger object
	DBGINIT(lgr, log, LOG_ENTRY_COUNT, LOG_ENTRY_LENGTH);

	ZeroCount      = 0;
	FltCount       = 0;
	FltFilter      = 0;
	FltFilterCount = 100; //100ms

	//turn off all delay timers
	for(i=0; i<DELAY_MAX; i++)
	{
		for(j=0; j<MAX_CHANNELS; j++)
		{
			IODelaySec[i][j] = -0.5; //Stoped
			IODelayBit[i][j] = 0;
		}
	}

	ZeroFlag       = 0;
	MasterMode     = STOP_MODE;
	//Screen.DoneVis = 1;
	qc[0].QCDoneVis = 1;
	qc[1].QCDoneVis = 1;

}

void _CYCLIC IO(void)
{

	//Startup delay???
	if (StartUpInit < 10000)
	{
		StartUpInit += TK_CYCLE_TIME_counts;
	}

	//detect belt zero signal rising edge
	ioBeltZeroDetect();

	//process and filter flite signal
	ioFliteDetect();

	//generate delay timers using 1ms cycle time
	hopperDelayTimers();

	//Handle force DO-s in case feature gets activated by the host
	if(diagIsForceDOsActive()){
		diagForceDOs();
	}else{
		outfeed();
	}
}
//eof
```

### Program Logical/Simulation/simonly (ANSIC)

#### simonly.c - Implementation code
```c
#include <..\..\GlobalDef.h>
#include <..\..\GlobalDecl.h>
//#include "..\\..\\RecFIFO\\fifotest\\fifoif.h"
#include "..\\..\\bglib\\bgsprintf.h"
#include "..\\..\\bglib\\bgsprintf.c"

static BOOL simIsProductAtInfeedWeigh()
{
	if(((MasterMode == RUN_MODE) || (MasterMode == FILL_MODE))&& (App[0].Hopper.State == APP4_FILL) ){
		return 1;
	}else{
		return 0;
	}
}

static BOOL simIsProductAtOutfeedWeigh()
{
	if((MasterMode == RUN_MODE) /*&& (App[1].Hopper.State == APP4_FILL)*/ && (OutfeedDumped == 1)){
		return 1;
	}else{
		return 0;
	}
}

static void simonlySimulateInfeedWt()
{
	if( simIsProductAtInfeedWeigh() ){
		Sys[0].Raw_wt = 8000;
	}else{
		if((MasterMode == RUN_MODE) || (MasterMode == FILL_MODE)){
			Sys[0].Raw_wt = 0;
		}
	}
}

static void simonlySimulateOutfeedWt()
{
	if( simIsProductAtOutfeedWeigh() ){
		Sys[1].Raw_wt = 2000;
	}else{
		if((MasterMode == RUN_MODE)){
			Sys[1].Raw_wt = 0;
		}
	}
}

static void simonlySimulateZeroFlag()
{
static int zeroFlagCounter;
static int zeroFlagState;

	//if BeltClutch is off > no updates / changes to the zero flag states
	if(!BeltClutch)
		return;

	switch(zeroFlagState){
		case 0:
			if(zeroFlagCounter++ > 1500){
				zeroFlagState = 1;
				zeroFlagCounter = 0;
				ZeroFlag = 1;
			}
		break;
		case 1:
			if(zeroFlagCounter++ > 5){
				zeroFlagState = 0;
				zeroFlagCounter = 0;
				ZeroFlag = 0;
			}
		break;
	}

}

void _INIT simonlyINIT(void)
{
	/* TODO: Add code here */

	//Overrid UDP Client operation settings (Use HMI if needed)
	//gUdpSystemCfg.udpClientMode = 1;//continues mode
	gUdpSystemCfg.udpClientUpdateRate = 5;//[Hz]
	strcpy(gUdpSystemCfg.udpRemoteHostIpAddress.text, "127.0.0.1");
	gUdpClient.clientIf.iTaskCycleTimeXms = 10;//udp client runs under 10ms cycle time

}

void _CYCLIC simonlyCYCLIC(void)
{
	/* TODO: Add code here */
	simonlySimulateInfeedWt();
	simonlySimulateOutfeedWt();
	simonlySimulateZeroFlag();

}
```

### Package Logical/HMI - HMI screens 

- Visualisation Logical/HMI/WSVGA (not shown)

### Package Logical/appConfigAndRecipes - application configuration and recipes

### appRecipe.typ - Global types - recipes - application level - CHANGE AS NEEDED
```iecst
(********************************************************************
 * COPYRIGHT --
 ********************************************************************
 * Package: paiConfigAndRecipes
 * File: appConfig.typ
 * Author: goran_2
 * Created: August 06, 2011
 ********************************************************************
 * Data types of package ConfigAndRecipes
 ********************************************************************)
(*==================================================================*)
(*Application recipe structure. Do not change the type name! Change content as needed.*)
(*==================================================================*)

TYPE
	cfgMachineRecipe_typ : 	STRUCT  (*Recipe structure*)
		name : STRING[126]; (*Recipe name*)
		author : STRING[31];
		dateLastSaved : STRING[31];
	END_STRUCT;
END_TYPE

(*######################################################*)
(*Below define type paiRecipeApp_typ MUST BE PRESENT!*)
(*ADD APPLICATION SPECIFIC MEMBERS AS NEEDED*)
(*######################################################*)

TYPE
	paiRecipeApp_typ : 	STRUCT  (*Recipe strucuture. DO NOT CHANGE.*)
		info : cfgMachineRecipe_typ; (*Active recipe*)
	END_STRUCT;
END_TYPE
```

### Program Logical/appConfigAndRecipes/appCfgRec (ANSIC) - app Config and Recipe Service (TK#8)

#### appCfgRec.var
```iecst
VAR
	fileRWBuffer : STRING[50000] := '';
	cfgFilename : STRING[63] := '';
END_VAR
VAR RETAIN
	gMagicRecipe : UDINT := 0;
END_VAR
```

#### paiPVSerDesMgrConfigure.c - Generic implementation code for the application's file storage service
```c
/********************************************************************
 * COPYRIGHT -- piedmont
 ********************************************************************
 * Program: cfgFS
 * File: cfgFS.c
 * Author: admin
 * Created: Jan 20, 2014
 ********************************************************************
 * Implementation of program cfgFS
 ********************************************************************/

#include <bur/plctypes.h>

#ifdef _DEFAULT_INCLUDES
 #include <AsDefault.h>
#endif

#include "../../paiComponents/bglib/bgPVSerialize.h"
#include "../appCfgRecDefault.h"
#include "../../paiComponents/paiFileService/paiPVSerDesMgr.h"
#include "../../paiComponents/paiFileService/paiFSInterface.h"
#include "../../paiComponents/paiFileService/paiFS/paiFile.h"

void gConfigAppDefaults();
void gPalletCfgDefaults();

/*
###############################################################################
PAI_CONFIGURATION_SECTION
Code below allows configuration of the PV serialization / deserialization
manager.
###############################################################################
*/
#warning "pai Configuration: Serialization/Deserialization"

void paiPVSerDesMgrConfigure()
{
	int itemIndex = 0;

	gPVSerDesMgr.pPaiFS = (UDINT)&paiFS;

	//add items as needed
	itemIndex = 0;
	brsstrcpy((UDINT)gPVSerDesMgr.pvItems[itemIndex].iPVName, (UDINT)"gConfigApp");
	brsstrcpy((UDINT)gPVSerDesMgr.pvItems[itemIndex].iDevicename, (UDINT)PAI_FS_DEVICE_CFG);
	brsstrcpy((UDINT)gPVSerDesMgr.pvItems[itemIndex].iFilename, (UDINT)"gConfigApp.txt");
	gPVSerDesMgr.pvItems[itemIndex].pPV = (UDINT)&gConfigApp;
	gPVSerDesMgr.pvItems[itemIndex].iPVSize = sizeof(gConfigApp);
	gPVSerDesMgr.pvItems[itemIndex].pFilebuffer = (UDINT)&fileRWBuffer[0];
	gPVSerDesMgr.pvItems[itemIndex].iFilebufferSize = sizeof(fileRWBuffer);
	gPVSerDesMgr.pvItems[itemIndex].pCallbackSer = (UDINT)paiCBWriteFileSerPV;
	gPVSerDesMgr.pvItems[itemIndex].pCallbackDes = (UDINT)paiCBReadFileDesPV;
	gPVSerDesMgr.pvItems[itemIndex].pCallbackDefault = (UDINT)gConfigAppDefaults;
	//Option: HMI interaction with PV read/write/changed; Allows PV changes to be accepted/rejected
	gPVSerDesMgr.pvItems[itemIndex].optPtrHMIData = &gSerDesHMI_gConfigApp;
	//Option: Monitor PV changes
	gPVSerDesMgr.pvItems[itemIndex].optChangeMonitor.iChngEnable = 1;
	gPVSerDesMgr.pvItems[itemIndex].optChangeMonitor.pChangeMonitorMem = &gSerDesMem_gConfigApp;
	gPVSerDesMgr.pvItems[itemIndex].optChangeMonitor.iChangeMonitorMemSize = sizeof(gSerDesMem_gConfigApp);
	//Option: Init PV at Power Up
	gPVSerDesMgr.pvItems[itemIndex].optInitAtPowerUp.iPowerUpConfig = PAI_FS_SERDESMGR_PWRUP_DFLT_fRD;
	gPVSerDesMgr.pvItems[itemIndex].optInitAtPowerUp.iTestData = 0x55555555;
	gPVSerDesMgr.pvItems[itemIndex].optInitAtPowerUp.pTestDataStorage = &gConfigApp.magicNumber;

	//add items as needed
	itemIndex = 1;
	brsstrcpy((UDINT)gPVSerDesMgr.pvItems[itemIndex].iPVName, (UDINT)"gPaiConfigSys");
	brsstrcpy((UDINT)gPVSerDesMgr.pvItems[itemIndex].iDevicename, (UDINT)PAI_FS_DEVICE_CFG);
	brsstrcpy((UDINT)gPVSerDesMgr.pvItems[itemIndex].iFilename, (UDINT)"gPaiConfigSys.txt");
	gPVSerDesMgr.pvItems[itemIndex].pPV = (UDINT)&gPaiConfigSys;
	gPVSerDesMgr.pvItems[itemIndex].iPVSize = sizeof(gPaiConfigSys);
	gPVSerDesMgr.pvItems[itemIndex].pFilebuffer = (UDINT)&fileRWBuffer[0];
	gPVSerDesMgr.pvItems[itemIndex].iFilebufferSize = sizeof(fileRWBuffer);
	gPVSerDesMgr.pvItems[itemIndex].pCallbackSer = (UDINT)paiCBWriteFileSerPV;
	gPVSerDesMgr.pvItems[itemIndex].pCallbackDes = (UDINT)paiCBReadFileDesPV;

	//add items as needed
	itemIndex = 2;
	brsstrcpy((UDINT)gPVSerDesMgr.pvItems[itemIndex].iPVName, (UDINT)"gLayerEditor");
	brsstrcpy((UDINT)gPVSerDesMgr.pvItems[itemIndex].iDevicename, (UDINT)PAI_FS_DEVICE_REC_LAYER);
	brsstrcpy((UDINT)gPVSerDesMgr.pvItems[itemIndex].iFilename, (UDINT)"recLayer.txt");
	gPVSerDesMgr.pvItems[itemIndex].pPV = (UDINT)&gLayerEditor;
	gPVSerDesMgr.pvItems[itemIndex].iPVSize = sizeof(gLayerEditor);
	gPVSerDesMgr.pvItems[itemIndex].pFilebuffer = (UDINT)&fileRWBuffer[0];
	gPVSerDesMgr.pvItems[itemIndex].iFilebufferSize = sizeof(fileRWBuffer);
	gPVSerDesMgr.pvItems[itemIndex].pCallbackSer = (UDINT)paiCBWriteFileSerPV;
	gPVSerDesMgr.pvItems[itemIndex].pCallbackDes = (UDINT)paiCBReadFileDesPV;
	gPVSerDesMgr.pvItems[itemIndex].pCallbackDefault = (UDINT)0;
	//Option: HMI interaction with PV read/write/changed; Allows PV changes to be accepted/rejected
	//gPVSerDesMgr.pvItems[itemIndex].optPtrHMIData = &gSerDesHMI_gConfigApp;
	//Option: Monitor PV changes
	gPVSerDesMgr.pvItems[itemIndex].optChangeMonitor.iChngEnable = 1;
	gPVSerDesMgr.pvItems[itemIndex].optChangeMonitor.pChangeMonitorMem = &gSerDesMem_gLayerEditor;
	gPVSerDesMgr.pvItems[itemIndex].optChangeMonitor.iChangeMonitorMemSize = sizeof(gSerDesMem_gLayerEditor);
	//Option: Init PV at Power Up
	gPVSerDesMgr.pvItems[itemIndex].optInitAtPowerUp.iPowerUpConfig = PAI_FS_SERDESMGR_PWRUP_DFLT_fRD;
	gPVSerDesMgr.pvItems[itemIndex].optInitAtPowerUp.iTestData = 0x55555555;
	gPVSerDesMgr.pvItems[itemIndex].optInitAtPowerUp.pTestDataStorage = &gDummy;

	//add items as needed
	itemIndex = 3;
	brsstrcpy((UDINT)gPVSerDesMgr.pvItems[itemIndex].iPVName, (UDINT)"gPallete.palCfg");
	brsstrcpy((UDINT)gPVSerDesMgr.pvItems[itemIndex].iDevicename, (UDINT)PAI_FS_DEVICE_REC_PALLETE);
	brsstrcpy((UDINT)gPVSerDesMgr.pvItems[itemIndex].iFilename, (UDINT)"recPallete.txt");
	gPVSerDesMgr.pvItems[itemIndex].pPV = (UDINT)&gPallete.palCfg;
	gPVSerDesMgr.pvItems[itemIndex].iPVSize = sizeof(gPallete.palCfg);
	gPVSerDesMgr.pvItems[itemIndex].pFilebuffer = (UDINT)&fileRWBuffer[0];
	gPVSerDesMgr.pvItems[itemIndex].iFilebufferSize = sizeof(fileRWBuffer);
	gPVSerDesMgr.pvItems[itemIndex].pCallbackSer = (UDINT)paiCBWriteFileSerPV;
	gPVSerDesMgr.pvItems[itemIndex].pCallbackDes = (UDINT)paiCBReadFileDesPV;
	gPVSerDesMgr.pvItems[itemIndex].pCallbackDefault = (UDINT)gPalletCfgDefaults;
	//Option: HMI interaction with PV read/write/changed; Allows PV changes to be accepted/rejected
	gPVSerDesMgr.pvItems[itemIndex].optPtrHMIData = &gSerDesHMI_gPalletCfg;
	//Option: Monitor PV changes
	gPVSerDesMgr.pvItems[itemIndex].optChangeMonitor.iChngEnable = 1;
	gPVSerDesMgr.pvItems[itemIndex].optChangeMonitor.pChangeMonitorMem = &gSerDesMem_gPallete_palCfg;
	gPVSerDesMgr.pvItems[itemIndex].optChangeMonitor.iChangeMonitorMemSize = sizeof(gSerDesMem_gPallete_palCfg);
	//Option: Init PV at Power Up
	gPVSerDesMgr.pvItems[itemIndex].optInitAtPowerUp.iPowerUpConfig = PAI_FS_SERDESMGR_PWRUP_DFLT_fRD;
	gPVSerDesMgr.pvItems[itemIndex].optInitAtPowerUp.iTestData = 0x55555555;
	//gPVSerDesMgr.pvItems[itemIndex].optInitAtPowerUp.pTestDataStorage = &gPallete.palCfg.magicNumber;
	gPVSerDesMgr.pvItems[itemIndex].optInitAtPowerUp.pTestDataStorage = &gMagicRecipe;

	//add items as needed
	itemIndex = 4;
	brsstrcpy((UDINT)gPVSerDesMgr.pvItems[itemIndex].iPVName, (UDINT)"gLayer_L0");
	brsstrcpy((UDINT)gPVSerDesMgr.pvItems[itemIndex].iDevicename, (UDINT)PAI_FS_DEVICE_REC_LAYER);
	brsstrcpy((UDINT)gPVSerDesMgr.pvItems[itemIndex].iFilename, (UDINT)"recLayer.txt");
	gPVSerDesMgr.pvItems[itemIndex].pPV = (UDINT)&gLayer_L0;
	gPVSerDesMgr.pvItems[itemIndex].iPVSize = sizeof(gLayer_L0);
	gPVSerDesMgr.pvItems[itemIndex].pFilebuffer = (UDINT)&fileRWBuffer[0];
	gPVSerDesMgr.pvItems[itemIndex].iFilebufferSize = sizeof(fileRWBuffer);
	gPVSerDesMgr.pvItems[itemIndex].pCallbackSer = (UDINT)paiCBWriteFileSerPV;
	gPVSerDesMgr.pvItems[itemIndex].pCallbackDes = (UDINT)paiCBReadFileDesPV;
	gPVSerDesMgr.pvItems[itemIndex].pCallbackDefault = (UDINT)0;
	//Option: HMI interaction with PV read/write/changed; Allows PV changes to be accepted/rejected
	//gPVSerDesMgr.pvItems[itemIndex].optPtrHMIData = &gSerDesHMI_gConfigApp;
	//Option: Monitor PV changes
	//gPVSerDesMgr.pvItems[itemIndex].optChangeMonitor.iChngEnable = 1;
	//gPVSerDesMgr.pvItems[itemIndex].optChangeMonitor.pChangeMonitorMem = &gSerDesMem_gLayerEditor;
	//gPVSerDesMgr.pvItems[itemIndex].optChangeMonitor.iChangeMonitorMemSize = sizeof(gSerDesMem_gLayerEditor);
	//Option: Init PV at Power Up
	//gPVSerDesMgr.pvItems[itemIndex].optInitAtPowerUp.iPowerUpConfig = PAI_FS_SERDESMGR_PWRUP_DFLT_fRD;
	//gPVSerDesMgr.pvItems[itemIndex].optInitAtPowerUp.iTestData = 0x55555555;
	//gPVSerDesMgr.pvItems[itemIndex].optInitAtPowerUp.pTestDataStorage = &gDummy;

	//add items as needed
	itemIndex = 5;
	brsstrcpy((UDINT)gPVSerDesMgr.pvItems[itemIndex].iPVName, (UDINT)"gLayer_L1");
	brsstrcpy((UDINT)gPVSerDesMgr.pvItems[itemIndex].iDevicename, (UDINT)PAI_FS_DEVICE_REC_LAYER);
	brsstrcpy((UDINT)gPVSerDesMgr.pvItems[itemIndex].iFilename, (UDINT)"recLayer.txt");
	gPVSerDesMgr.pvItems[itemIndex].pPV = (UDINT)&gLayer_L1;
	gPVSerDesMgr.pvItems[itemIndex].iPVSize = sizeof(gLayer_L1);
	gPVSerDesMgr.pvItems[itemIndex].pFilebuffer = (UDINT)&fileRWBuffer[0];
	gPVSerDesMgr.pvItems[itemIndex].iFilebufferSize = sizeof(fileRWBuffer);
	gPVSerDesMgr.pvItems[itemIndex].pCallbackSer = (UDINT)paiCBWriteFileSerPV;
	gPVSerDesMgr.pvItems[itemIndex].pCallbackDes = (UDINT)paiCBReadFileDesPV;
	gPVSerDesMgr.pvItems[itemIndex].pCallbackDefault = (UDINT)0;
	//Option: HMI interaction with PV read/write/changed; Allows PV changes to be accepted/rejected
	//gPVSerDesMgr.pvItems[itemIndex].optPtrHMIData = &gSerDesHMI_gConfigApp;
	//Option: Monitor PV changes
	//gPVSerDesMgr.pvItems[itemIndex].optChangeMonitor.iChngEnable = 1;
	//gPVSerDesMgr.pvItems[itemIndex].optChangeMonitor.pChangeMonitorMem = &gSerDesMem_gLayerEditor;
	//gPVSerDesMgr.pvItems[itemIndex].optChangeMonitor.iChangeMonitorMemSize = sizeof(gSerDesMem_gLayerEditor);
	//Option: Init PV at Power Up
	//gPVSerDesMgr.pvItems[itemIndex].optInitAtPowerUp.iPowerUpConfig = PAI_FS_SERDESMGR_PWRUP_DFLT_fRD;
	//gPVSerDesMgr.pvItems[itemIndex].optInitAtPowerUp.iTestData = 0x55555555;
	//gPVSerDesMgr.pvItems[itemIndex].optInitAtPowerUp.pTestDataStorage = &gDummy;

	//Set number of active items for PVSerDes Mgr
	gPVSerDesMgr.iItemCount = itemIndex + 1;

	//invoke paiSerDesMgr init routine
	paiPVSerDesMgrInit(&gPVSerDesMgr);
}
//EOF
```

- bgPVSerialize.c (reference to Logical/paiComponents/bglib/bgPVSerialize.c)

- bgstring.c (reference to Logical/paiComponents/bglib/bgstring.c)

- paiFSInterface.c (reference to Logical/paiComponents/paiFileService/paiFSInterface.c)

- Defaults_gConfigApp.c (reference to Logical/Globals/Defaults_gConfigApp.c)

### ParameterDownload.typ
```iecst
(********************************************************************
 * COPYRIGHT --
 ********************************************************************
 * Program: S44param
 * File: S44param.typ
 * Author: scoccimaroj
 * Created: July 15, 2010
 ********************************************************************
 * Local data types of program S44param
 ********************************************************************)

TYPE
	X64ParamRead_typ : 	STRUCT
		pDevice : STRING[30]; (*Device string of the inverter*)
		FileDevice : STRING[20]; (*Device string for writing the csv file.*)
		FilePath : STRING[30]; (*CSV File path*)
		CsvFileName : STRING[50]; (*name of the csv file*)
		Parameters : ARRAY[0..NUM_OF_X64PAR]OF ASIOACCPar_typ;
	END_STRUCT;
	S44ParamRead_typ : 	STRUCT
		pDevice : STRING[30]; (*Device string of the inverter*)
		FileDevice : STRING[20]; (*Device string for writing the csv file.*)
		FilePath : STRING[30]; (*CSV File path*)
		CsvFileName : STRING[50]; (*name of the csv file*)
		Parameters : ARRAY[0..NUM_OF_S44PAR]OF ASIOACCPar_typ;
	END_STRUCT;
	ASIOACCPar_typ : 	STRUCT
		ChannelName : STRING[15]; (*Device string of the inverter*)
		Data : UDINT;
	END_STRUCT;
	P84ParamRead_typ : 	STRUCT
		pDevice : STRING[30]; (*Device string of the inverter*)
		FileDevice : STRING[20]; (*Device string for writing the csv file.*)
		FilePath : STRING[30]; (*CSV File path*)
		CsvFileName : STRING[50]; (*name of the csv file*)
		NodeNr : USINT; (*node number of the inverter on the EPL network*)
		Parameters : ARRAY[0..NUM_OF_P84PAR]OF EPLPar_typ;
	END_STRUCT;
	EPLPar_typ : 	STRUCT
		Index : UINT;
		Subindex : USINT;
		Data : UDINT;
		Code : STRING[5];
	END_STRUCT;
	P74ParamRead_typ : 	STRUCT
		pDevice : STRING[30]; (*Device string of the inverter*)
		FileDevice : STRING[20]; (*Device string for writing the csv file.*)
		FilePath : STRING[30]; (*CSV File path*)
		CsvFileName : STRING[50]; (*name of the csv file*)
		NodeNr : USINT; (*node number of the inverter on the EPL network*)
		Parameters : ARRAY[0..NUM_OF_P74PAR]OF EPLPar_typ;
	END_STRUCT;
END_TYPE
```

### ParameterDownload.var
```iecst
(********************************************************************
 * COPYRIGHT --
 ********************************************************************
 * Program: S44param
 * File: S44param.var
 * Author: scoccimaroj
 * Created: July 15, 2010
 ********************************************************************
 * Local variables of program S44param
 ********************************************************************)
VAR
	P84ParRead : P84ParamRead_typ; (*Variable used to store parameter data*)
	X64ParRead : X64ParamRead_typ; (*Holds the information for the X64 parameters that are read*)
	S44ParRead : S44ParamRead_typ; (*Holds the information for the X64 parameters that are read*)
	P74ParRead : P74ParamRead_typ; (*Variable used to store parameter data*)
END_VAR
(*Constants*)
VAR CONSTANT
	NUM_OF_S44PAR : UINT := 123; (*Number of x64 parameters*)
	NUM_OF_X64PAR : UINT := 138; (*Number of x64 parameters*)
	NUM_OF_P74PAR : UINT := 836; (*Number of P84 parameters in the IO configuration screen*)
	NUM_OF_P84PAR : UINT := 362; (*Number of P84 parameters in the IO configuration screen*)
END_VAR
```

### Library Logical/ParameterDownload/CSV_File (IEC, version 2.01.8)
Depends on: AsMath, AsMem, AsString, FileIO, runtime, standard, sys_lib, astime

#### CSV_CheckFile.ab
```automation-basic
FUNCTION_BLOCK CSV_CheckFile
(********************************************************************
 * COPYRIGHT -- Bernecker + Rainer Industrie Elektronik GmbH
 ********************************************************************
 * Library: CSV_File
 * File: CSV_CheckFile.ab
 * Author: kreidlm
 * Created: November 29, 2006
 ********************************************************************
 * Implementation of library CSV_File
 ********************************************************************)

CharPerCyclic = CharPerCyclic

R_TRIG_0.CLK = enable
R_TRIG_0 FUB R_TRIG()

select fileCheckStep of
	;##########################################################################################
    state WAIT
	;##########################################################################################

        when (R_TRIG_0.CLK = 1) and ( (pFileName = 0) or (pDevice = 0) or (pStructSizes = 0) or (pVersion = 0) or (pFileBuffer = 0) ) do
            status = ERROR_INPUT_POINTER_ERR;
       	next WAIT

        when (R_TRIG_0.CLK = 1) do
            status = 65535
            statusInternal = 0
            fileError = 0
            lineCnt = 0
            maxLenLine = SIZEOF(lineBuf)-1
            versionFound = 0
            cntSizesFound = 0
            memset(adr(SizesFound), 0, SIZEOF(SizesFound))
            strcpy(adr(verSignificationStr),"// V")
            strcpy(adr(sizeSignificationStr), "// Structure Size: ")
            strcpy(adr(fileVersionStr), "")
        next FOPEN

	;##########################################################################################
    state FOPEN
	;##########################################################################################
    	FOpen.enable = 1
        FOpen.pDevice  = pDevice
        FOpen.pFile = pFileName
        FOpen.mode = 2

        FOpen FUB FileOpen()
        fileIdent = FOpen.ident
        statusInternal = FOpen.status

        when (statusInternal = 0) and (FOpen.filelen < FileBufferSize) do
            memset(pFileBuffer, 0 , FileBufferSize)
            pChar access (pFileBuffer+FOpen.filelen)
            pChar = 0 (* Terminierung ans Ende des Filebuffers*)
            status = 65535
        next FREAD
        (* File zu gross für Buffer *)
        when (statusInternal = 0) and (FOpen.filelen >= FileBufferSize) do
        	statusInternal = ERROR_CHECKFILEBUFFER_TOO_SMALL
            status = statusInternal
        next WAIT
        when ((statusInternal <> 0) and (statusInternal <> 65535)) do
            if (statusInternal = fiERR_SYSTEM) then
                fileError = FileIoGetSysError()
            endif
            status = statusInternal
        next WAIT

	;##########################################################################################
    state FREAD
	;##########################################################################################
         FRead.enable = 1
         FRead.ident = fileIdent
         FRead.offset = 0
         FRead.pDest = pFileBuffer
         FRead.len = FOpen.filelen

         FRead FUB FileRead()
         statusInternal = FRead.status

         when (statusInternal = 0) do
            loop fileOffset = 0 to (FOpen.filelen-1) do
                pChar access (pFileBuffer+fileOffset)
                if (pChar = 10) then (* LF *)
            	    pChar = 0 (* durch Terminator ersetzen *)
                    lineCnt = lineCnt + 1
                endif
   	        endloop
            fileOffset = pFileBuffer
            status = 65535
         next FCLOSE
         when ((statusInternal <> 0) and (statusInternal <> 65535)) do
            if (statusInternal = fiERR_SYSTEM) then
                fileError = FileIoGetSysError()
            endif
            status = statusInternal
         next WAIT

	;##########################################################################################
	state FCLOSE
	;##########################################################################################
    	FClose.enable = 1
        FClose.ident = fileIdent

        FClose FUB FileClose()
        statusInternal = FClose.status

        when (statusInternal = 0) do
        	status = 65535
        next FCHECK
        when ((statusInternal <> 0) and (statusInternal <> 65535)) do
            if (statusInternal = fiERR_SYSTEM) then
                fileError = FileIoGetSysError()
            endif
            status = statusInternal
        next WAIT

	;##########################################################################################
    state FCHECK
	;##########################################################################################
        when (1=1) do
            if (lineCnt > 0) then
                ixLineMax = lineCnt - 1
            else
            	ixLineMax = 0
            endif
            ;Filebuffer parsen
            loop ixLine = 0 to ixLineMax do
                if (strlen(fileOffset) <= maxLenLine ) then
                    strcpy(adr(lineBuf), fileOffset)
                    if ((FIND(lineBuf, verSignificationStr) = 1) and (versionFound = 0)) then
                        fileVersionStr = MID(lineBuf, strlen(pVersion), strlen(adr(verSignificationStr)))
                        versionFound = 1
                    endif
                    if ((FIND(lineBuf, sizeSignificationStr) = 1) and (cntSizesFound < NumOfStruct)) then
                        SizesFound[cntSizesFound] = atoi(adr(lineBuf) + strlen(adr(sizeSignificationStr)))
                        cntSizesFound = cntSizesFound + 1
                    endif
                endif
                fileOffset = fileOffset + strlen(fileOffset) + 1
            endloop
            ;Auswertung
            if (strcmp(adr(fileVersionStr), pVersion) <> 0) then
                statusInternal = ERROR_VERSION_MISMATCH
            endif
            if (cntSizesFound <> NumOfStruct) then
        	    statusInternal = ERROR_NUM_OF_STRUCT_MISMATCH
            endif
       	    if (NumOfStruct > 0) then
                loop ixCmp = 0 to (NumOfStruct-1) do
                    pSize access (pStructSizes + ixCmp*SIZEOF(SizesFound[0]))
                    if (SizesFound[ixCmp] <> pSize) then
                        statusInternal = ERROR_SIZE_MISMATCH
                    endif
                    exitif (statusInternal = ERROR_SIZE_MISMATCH)
                endloop
            else
                statusInternal = ERROR_NUM_OF_STRUCT_MISMATCH
            endif
            status = statusInternal
      	next WAIT

endselect
END_FUNCTION_BLOCK
```
